LIN {X 0,Y 390.118,Z 257.391,A -85,B 0,C 180,E1 -11800.378,E2 -11800.378} C_VEL
LIN {X 0,Y 390.108,Z 257.393,A -85,B 0,C 180,E1 -11803.544,E2 -11803.544} C_VEL
LIN {X 0,Y 390.089,Z 257.395,A -85,B 0,C 180,E1 -11807.311,E2 -11807.311} C_VEL
LIN {X 0,Y 390.049,Z 257.395,A -85,B 0,C 180,E1 -11811.122,E2 -11811.122} C_VEL
LIN {X 0,Y 390.027,Z 257.402,A -85,B 0,C 180,E1 -11814.484,E2 -11814.484} C_VEL
LIN {X 0,Y 390.06,Z 257.399,A -85,B 0,C 180,E1 -11818.029,E2 -11818.029} C_VEL
LIN {X 0,Y 389.97,Z 257.406,A -85,B 0,C 180,E1 -11820.774,E2 -11820.774} C_VEL
LIN {X 0,Y 389.303,Z 257.492,A -85,B 0,C 180,E1 -11821.636,E2 -11821.636} C_VEL
LIN {X 0,Y 386.453,Z 257.843,A -85,B 0,C 180,E1 -11823.037,E2 -11823.037} C_VEL
LIN {X 0,Y 384.048,Z 258.147,A -85,B 0,C 180,E1 -11824.17,E2 -11824.17} C_VEL
LIN {X 0,Y 383.025,Z 258.271,A -85,B 0,C 180,E1 -11825.046,E2 -11825.046} C_VEL
LIN {X 0,Y 382.946,Z 258.281,A -85,B 0,C 180,E1 -11825.343,E2 -11825.343} C_VEL
LIN {X 0,Y 382.958,Z 258.279,A -85,B 0,C 180,E1 -11828.605,E2 -11828.605} C_VEL
LIN {X 0,Y 382.999,Z 258.276,A -85,B 0,C 180,E1 -11831.344,E2 -11831.344} C_VEL
LIN {X 0,Y 383.025,Z 258.271,A -85,B 0,C 180,E1 -11834.32,E2 -11834.32} C_VEL
LIN {X 0,Y 383.033,Z 258.272,A -85,B 0,C 180,E1 -11837.255,E2 -11837.255} C_VEL
LIN {X 0,Y 382.974,Z 258.276,A -85,B 0,C 180,E1 -11840.42,E2 -11840.42} C_VEL
LIN {X 0,Y 382.987,Z 258.276,A -85,B 0,C 180,E1 -11844.05,E2 -11844.05} C_VEL
LIN {X 0,Y 382.952,Z 258.283,A -85,B 0,C 180,E1 -11847.585,E2 -11847.585} C_VEL
LIN {X 0,Y 382.96,Z 258.278,A -85,B 0,C 180,E1 -11850.306,E2 -11850.306} C_VEL
LIN {X 0,Y 383.052,Z 258.267,A -85,B 0,C 180,E1 -11854.028,E2 -11854.028} C_VEL
LIN {X 0,Y 382.969,Z 258.28,A -85,B 0,C 180,E1 -11857.341,E2 -11857.341} C_VEL
LIN {X 0,Y 383.035,Z 258.274,A -85,B 0,C 180,E1 -11860.723,E2 -11860.723} C_VEL
LIN {X 0,Y 383.059,Z 258.266,A -85,B 0,C 180,E1 -11864.033,E2 -11864.033} C_VEL
LIN {X 0,Y 383.119,Z 258.259,A -85,B 0,C 180,E1 -11867.29,E2 -11867.29} C_VEL
LIN {X 0,Y 383.128,Z 258.263,A -85,B 0,C 180,E1 -11870.504,E2 -11870.504} C_VEL
LIN {X 0,Y 383.248,Z 258.243,A -85,B 0,C 180,E1 -11873.69,E2 -11873.69} C_VEL
LIN {X 0,Y 383.37,Z 258.229,A -85,B 0,C 180,E1 -11877.905,E2 -11877.905} C_VEL
LIN {X 0,Y 383.366,Z 258.233,A -85,B 0,C 180,E1 -11882.107,E2 -11882.107} C_VEL
LIN {X 0,Y 383.229,Z 258.249,A -85,B 0,C 180,E1 -11886.323,E2 -11886.323} C_VEL
LIN {X 0,Y 383.14,Z 258.257,A -85,B 0,C 180,E1 -11889.508,E2 -11889.508} C_VEL
LIN {X 0,Y 383.127,Z 258.26,A -85,B 0,C 180,E1 -11893.541,E2 -11893.541} C_VEL
LIN {X 0,Y 383.056,Z 258.269,A -85,B 0,C 180,E1 -11897.439,E2 -11897.439} C_VEL
LIN {X 0,Y 383.021,Z 258.271,A -85,B 0,C 180,E1 -11900.647,E2 -11900.647} C_VEL
LIN {X 0,Y 383.013,Z 258.276,A -85,B 0,C 180,E1 -11903.814,E2 -11903.814} C_VEL
LIN {X 0,Y 382.976,Z 258.281,A -85,B 0,C 180,E1 -11907.313,E2 -11907.313} C_VEL
LIN {X 0,Y 382.989,Z 258.277,A -85,B 0,C 180,E1 -11910.923,E2 -11910.923} C_VEL
LIN {X 0,Y 383.021,Z 258.276,A -85,B 0,C 180,E1 -11914.673,E2 -11914.673} C_VEL
LIN {X 0,Y 383.005,Z 258.278,A -85,B 0,C 180,E1 -11917.906,E2 -11917.906} C_VEL
LIN {X 0,Y 383.229,Z 259.82,A -85,B 0,C 180,E1 -11919.936,E2 -11919.936} C_VEL
LIN {X 0,Y 383.606,Z 262.486,A -85,B 0,C 180,E1 -11922.877,E2 -11922.877} C_VEL
LIN {X 0,Y 384.023,Z 265.533,A -85,B 0,C 180,E1 -11925.939,E2 -11925.939} C_VEL
LIN {X 0,Y 384.15,Z 268.607,A -85,B 0,C 180,E1 -11928.806,E2 -11928.806} C_VEL
LIN {X 0,Y 383.846,Z 272.282,A -85,B 0,C 180,E1 -11931.94,E2 -11931.94} C_VEL
LIN {X 0,Y 383.375,Z 276.85,A -85,B 0,C 180,E1 -11935.588,E2 -11935.588} C_VEL
LIN {X 0,Y 382.941,Z 281.501,A -85,B 0,C 180,E1 -11939.078,E2 -11939.078} C_VEL
LIN {X 0,Y 382.565,Z 286.485,A -85,B 0,C 180,E1 -11942.661,E2 -11942.661} C_VEL
LIN {X 0,Y 382.195,Z 291.542,A -85,B 0,C 180,E1 -11946.138,E2 -11946.138} C_VEL
LIN {X 0,Y 381.988,Z 297.019,A -85,B 0,C 180,E1 -11949.78,E2 -11949.78} C_VEL
LIN {X 0,Y 381.923,Z 299.239,A -85,B 0,C 180,E1 -11951.102,E2 -11951.102} C_VEL
LIN {X 0,Y 384.001,Z 309.515,A -85,B 0,C 180,E1 -11951.545,E2 -11951.545} C_VEL
LIN {X 0,Y 385.658,Z 318.988,A -85,B 0,C 180,E1 -11952.062,E2 -11952.062} C_VEL
LIN {X 0,Y 387.132,Z 329.109,A -85,B 0,C 180,E1 -11952.736,E2 -11952.736} C_VEL
LIN {X 0,Y 387.167,Z 334.549,A -85,B 0,C 180,E1 -11953.116,E2 -11953.116} C_VEL
LIN {X 0,Y 386.22,Z 345.46,A -85,B 0,C 180,E1 -11954.025,E2 -11954.025} C_VEL
LIN {X 0,Y 385.421,Z 354.407,A -85,B 0,C 180,E1 -11954.94,E2 -11954.94} C_VEL
LIN {X 0,Y 384.666,Z 363.303,A -85,B 0,C 180,E1 -11956.041,E2 -11956.041} C_VEL
LIN {X 0,Y 384.092,Z 370.167,A -85,B 0,C 180,E1 -11957.048,E2 -11957.048} C_VEL
LIN {X 0,Y 383.446,Z 376.37,A -85,B 0,C 180,E1 -11958.101,E2 -11958.101} C_VEL
LIN {X 0,Y 382.875,Z 382.911,A -85,B 0,C 180,E1 -11959.423,E2 -11959.423} C_VEL
LIN {X 0,Y 382.469,Z 387.414,A -85,B 0,C 180,E1 -11960.481,E2 -11960.481} C_VEL
LIN {X 0,Y 382.045,Z 392.908,A -85,B 0,C 180,E1 -11962.07,E2 -11962.07} C_VEL
LIN {X 0,Y 381.783,Z 397.235,A -85,B 0,C 180,E1 -11963.659,E2 -11963.659} C_VEL
LIN {X 0,Y 381.68,Z 399.603,A -85,B 0,C 180,E1 -11964.718,E2 -11964.718} C_VEL
LIN {X 0,Y 381.644,Z 401.403,A -85,B 0,C 180,E1 -11965.776,E2 -11965.776} C_VEL
LIN {X 0,Y 381.564,Z 403.848,A -85,B 0,C 180,E1 -11967.889,E2 -11967.889} C_VEL
LIN {X 0,Y 381.598,Z 404.437,A -85,B 0,C 180,E1 -11968.945,E2 -11968.945} C_VEL
LIN {X 0,Y 381.598,Z 404.437,A -85,B 0,C 180,E1 -11971.055,E2 -11971.055} C_VEL
LIN {X 0,Y 381.564,Z 403.848,A -85,B 0,C 180,E1 -11972.111,E2 -11972.111} C_VEL
LIN {X 0,Y 381.644,Z 401.403,A -85,B 0,C 180,E1 -11974.224,E2 -11974.224} C_VEL
LIN {X 0,Y 381.689,Z 398.553,A -85,B 0,C 180,E1 -11975.768,E2 -11975.768} C_VEL
LIN {X 0,Y 381.947,Z 394.463,A -85,B 0,C 180,E1 -11977.4,E2 -11977.4} C_VEL
LIN {X 0,Y 382.314,Z 389.331,A -85,B 0,C 180,E1 -11978.989,E2 -11978.989} C_VEL
LIN {X 0,Y 382.758,Z 384.067,A -85,B 0,C 180,E1 -11980.313,E2 -11980.313} C_VEL
LIN {X 0,Y 383.294,Z 377.746,A -85,B 0,C 180,E1 -11981.636,E2 -11981.636} C_VEL
LIN {X 0,Y 383.899,Z 371.793,A -85,B 0,C 180,E1 -11982.69,E2 -11982.69} C_VEL
LIN {X 0,Y 384.536,Z 364.863,A -85,B 0,C 180,E1 -11983.744,E2 -11983.744} C_VEL
LIN {X 0,Y 385.231,Z 356.678,A -85,B 0,C 180,E1 -11984.798,E2 -11984.798} C_VEL
LIN {X 0,Y 385.954,Z 348.163,A -85,B 0,C 180,E1 -11985.715,E2 -11985.715} C_VEL
LIN {X 0,Y 386.696,Z 339.445,A -85,B 0,C 180,E1 -11986.497,E2 -11986.497} C_VEL
LIN {X 0,Y 387.344,Z 331.917,A -85,B 0,C 180,E1 -11987.065,E2 -11987.065} C_VEL
LIN {X 0,Y 386.126,Z 321.842,A -85,B 0,C 180,E1 -11987.765,E2 -11987.765} C_VEL
LIN {X 0,Y 384.183,Z 310.483,A -85,B 0,C 180,E1 -11988.408,E2 -11988.408} C_VEL
LIN {X 0,Y 381.981,Z 299.866,A -85,B 0,C 180,E1 -11988.879,E2 -11988.879} C_VEL
LIN {X 0,Y 381.893,Z 299.048,A -85,B 0,C 180,E1 -11988.926,E2 -11988.926} C_VEL
LIN {X 0,Y 382.068,Z 294.919,A -85,B 0,C 180,E1 -11991.585,E2 -11991.585} C_VEL
LIN {X 0,Y 382.33,Z 289.843,A -85,B 0,C 180,E1 -11995.01,E2 -11995.01} C_VEL
LIN {X 0,Y 382.699,Z 284.821,A -85,B 0,C 180,E1 -11998.52,E2 -11998.52} C_VEL
LIN {X 0,Y 382.943,Z 281.501,A -85,B 0,C 180,E1 -12000.921,E2 -12000.921} C_VEL
LIN {X 0,Y 383.405,Z 276.573,A -85,B 0,C 180,E1 -12004.627,E2 -12004.627} C_VEL
LIN {X 0,Y 383.845,Z 272.283,A -85,B 0,C 180,E1 -12008.06,E2 -12008.06} C_VEL
LIN {X 0,Y 384.144,Z 268.607,A -85,B 0,C 180,E1 -12011.194,E2 -12011.194} C_VEL
LIN {X 0,Y 384.185,Z 266.644,A -85,B 0,C 180,E1 -12012.963,E2 -12012.963} C_VEL
LIN {X 0,Y 383.802,Z 263.652,A -85,B 0,C 180,E1 -12015.901,E2 -12015.901} C_VEL
LIN {X 0,Y 383.391,Z 260.995,A -85,B 0,C 180,E1 -12018.726,E2 -12018.726} C_VEL
LIN {X 0,Y 383.005,Z 258.278,A -85,B 0,C 180,E1 -12022.094,E2 -12022.094} C_VEL
LIN {X 0,Y 383.021,Z 258.276,A -85,B 0,C 180,E1 -12025.327,E2 -12025.327} C_VEL
LIN {X 0,Y 382.989,Z 258.277,A -85,B 0,C 180,E1 -12029.077,E2 -12029.077} C_VEL
LIN {X 0,Y 382.976,Z 258.281,A -85,B 0,C 180,E1 -12032.687,E2 -12032.687} C_VEL
LIN {X 0,Y 383.013,Z 258.276,A -85,B 0,C 180,E1 -12036.186,E2 -12036.186} C_VEL
LIN {X 0,Y 383.045,Z 258.268,A -85,B 0,C 180,E1 -12039.593,E2 -12039.593} C_VEL
LIN {X 0,Y 383.072,Z 258.265,A -85,B 0,C 180,E1 -12042.925,E2 -12042.925} C_VEL
LIN {X 0,Y 383.127,Z 258.26,A -85,B 0,C 180,E1 -12046.459,E2 -12046.459} C_VEL
LIN {X 0,Y 383.14,Z 258.257,A -85,B 0,C 180,E1 -12050.492,E2 -12050.492} C_VEL
LIN {X 0,Y 383.229,Z 258.249,A -85,B 0,C 180,E1 -12053.677,E2 -12053.677} C_VEL
LIN {X 0,Y 383.366,Z 258.233,A -85,B 0,C 180,E1 -12057.893,E2 -12057.893} C_VEL
LIN {X 0,Y 383.37,Z 258.229,A -85,B 0,C 180,E1 -12062.095,E2 -12062.095} C_VEL
LIN {X 0,Y 383.228,Z 258.245,A -85,B 0,C 180,E1 -12066.567,E2 -12066.567} C_VEL
LIN {X 0,Y 383.128,Z 258.263,A -85,B 0,C 180,E1 -12069.496,E2 -12069.496} C_VEL
LIN {X 0,Y 383.108,Z 258.264,A -85,B 0,C 180,E1 -12073.529,E2 -12073.529} C_VEL
LIN {X 0,Y 383.073,Z 258.269,A -85,B 0,C 180,E1 -12077.063,E2 -12077.063} C_VEL
LIN {X 0,Y 383.005,Z 258.275,A -85,B 0,C 180,E1 -12080.64,E2 -12080.64} C_VEL
LIN {X 0,Y 382.999,Z 258.274,A -85,B 0,C 180,E1 -12083.801,E2 -12083.801} C_VEL
LIN {X 0,Y 383.051,Z 258.267,A -85,B 0,C 180,E1 -12086.117,E2 -12086.117} C_VEL
LIN {X 0,Y 382.96,Z 258.278,A -85,B 0,C 180,E1 -12089.694,E2 -12089.694} C_VEL
LIN {X 0,Y 382.968,Z 258.278,A -85,B 0,C 180,E1 -12093.395,E2 -12093.395} C_VEL
LIN {X 0,Y 382.994,Z 258.276,A -85,B 0,C 180,E1 -12096.158,E2 -12096.158} C_VEL
LIN {X 0,Y 382.972,Z 258.278,A -85,B 0,C 180,E1 -12099.952,E2 -12099.952} C_VEL
LIN {X 0,Y 383.023,Z 258.273,A -85,B 0,C 180,E1 -12102.783,E2 -12102.783} C_VEL
LIN {X 0,Y 383.027,Z 258.271,A -85,B 0,C 180,E1 -12105.795,E2 -12105.795} C_VEL
LIN {X 0,Y 382.997,Z 258.275,A -85,B 0,C 180,E1 -12108.781,E2 -12108.781} C_VEL
LIN {X 0,Y 382.953,Z 258.285,A -85,B 0,C 180,E1 -12112.091,E2 -12112.091} C_VEL
LIN {X 0,Y 382.966,Z 258.278,A -85,B 0,C 180,E1 -12115.327,E2 -12115.327} C_VEL
LIN {X 0,Y 382.983,Z 258.281,A -85,B 0,C 180,E1 -12117.848,E2 -12117.848} C_VEL
LIN {X 0,Y 383.008,Z 258.277,A -85,B 0,C 180,E1 -12121.717,E2 -12121.717} C_VEL
LIN {X 0,Y 382.997,Z 258.274,A -85,B 0,C 180,E1 -12125.036,E2 -12125.036} C_VEL
LIN {X 0,Y 383.016,Z 258.271,A -85,B 0,C 180,E1 -12128.471,E2 -12128.471} C_VEL
LIN {X 0,Y 383.034,Z 258.274,A -85,B 0,C 180,E1 -12131.825,E2 -12131.825} C_VEL
LIN {X 0,Y 383.055,Z 258.272,A -85,B 0,C 180,E1 -12135.116,E2 -12135.116} C_VEL
LIN {X 0,Y 383.046,Z 258.271,A -85,B 0,C 180,E1 -12138.357,E2 -12138.357} C_VEL
LIN {X 0,Y 383.112,Z 258.465,A -85,B 0,C 180,E1 -12139.597,E2 -12139.597} C_VEL
LIN {X 0,Y 383.808,Z 260.603,A -85,B 0,C 180,E1 -12139.949,E2 -12139.949} C_VEL
LIN {X 0,Y 385.342,Z 262.607,A -85,B 0,C 180,E1 -12140.685,E2 -12140.685} C_VEL
LIN {X 0,Y 387.431,Z 263.893,A -85,B 0,C 180,E1 -12141.656,E2 -12141.656} C_VEL
LIN {X 0,Y 388.82,Z 264.575,A -85,B 0,C 180,E1 -12142.393,E2 -12142.393} C_VEL
LIN {X 0,Y 389.855,Z 266.733,A -85,B 0,C 180,E1 -12143.075,E2 -12143.075} C_VEL
LIN {X 0,Y 391.629,Z 268.873,A -85,B 0,C 180,E1 -12144.336,E2 -12144.336} C_VEL
LIN {X 0,Y 393.42,Z 270.078,A -85,B 0,C 180,E1 -12145.902,E2 -12145.902} C_VEL
LIN {X 0,Y 394.315,Z 270.312,A -85,B 0,C 180,E1 -12146.935,E2 -12146.935} C_VEL
LIN {X 0,Y 395.344,Z 270.546,A -85,B 0,C 180,E1 -12148.981,E2 -12148.981} C_VEL
LIN {X 0,Y 395.505,Z 270.523,A -85,B 0,C 180,E1 -12150,E2 -12150} C_VEL
LIN {X 0,Y 394.942,Z 270.448,A -85,B 0,C 180,E1 -12152.04,E2 -12152.04} C_VEL
LIN {X 0,Y 394.144,Z 270.274,A -85,B 0,C 180,E1 -12153.268,E2 -12153.268} C_VEL
LIN {X 0,Y 392.863,Z 269.796,A -85,B 0,C 180,E1 -12154.617,E2 -12154.617} C_VEL
LIN {X 0,Y 390.976,Z 268.254,A -85,B 0,C 180,E1 -12156.127,E2 -12156.127} C_VEL
LIN {X 0,Y 389.275,Z 265.68,A -85,B 0,C 180,E1 -12157.318,E2 -12157.318} C_VEL
LIN {X 0,Y 388.598,Z 264.268,A -85,B 0,C 180,E1 -12157.735,E2 -12157.735} C_VEL
LIN {X 0,Y 386.111,Z 263.182,A -85,B 0,C 180,E1 -12158.966,E2 -12158.966} C_VEL
LIN {X 0,Y 384.201,Z 261.281,A -85,B 0,C 180,E1 -12159.861,E2 -12159.861} C_VEL
LIN {X 0,Y 383.227,Z 259.103,A -85,B 0,C 180,E1 -12160.333,E2 -12160.333} C_VEL
LIN {X 0,Y 383.073,Z 258.269,A -85,B 0,C 180,E1 -12160.438,E2 -12160.438} C_VEL
LIN {X 0,Y 383.066,Z 258.269,A -85,B 0,C 180,E1 -12163.798,E2 -12163.798} C_VEL
LIN {X 0,Y 383.036,Z 258.273,A -85,B 0,C 180,E1 -12167.458,E2 -12167.458} C_VEL
LIN {X 0,Y 383.005,Z 258.276,A -85,B 0,C 180,E1 -12170.664,E2 -12170.664} C_VEL
LIN {X 0,Y 382.99,Z 258.276,A -85,B 0,C 180,E1 -12173.81,E2 -12173.81} C_VEL
LIN {X 0,Y 383,Z 258.273,A -85,B 0,C 180,E1 -12177.306,E2 -12177.306} C_VEL
LIN {X 0,Y 382.941,Z 258.281,A -85,B 0,C 180,E1 -12180.922,E2 -12180.922} C_VEL
LIN {X 0,Y 382.965,Z 258.28,A -85,B 0,C 180,E1 -12184.344,E2 -12184.344} C_VEL
LIN {X 0,Y 382.946,Z 258.281,A -85,B 0,C 180,E1 -12185.343,E2 -12185.343} C_VEL
LIN {X 0,Y 382.302,Z 258.367,A -85,B 0,C 180,E1 -12186.221,E2 -12186.221} C_VEL
LIN {X 0,Y 379.489,Z 258.724,A -85,B 0,C 180,E1 -12187.65,E2 -12187.65} C_VEL
LIN {X 0,Y 377.089,Z 259.023,A -85,B 0,C 180,E1 -12188.804,E2 -12188.804} C_VEL
LIN {X 0,Y 376.043,Z 259.147,A -85,B 0,C 180,E1 -12189.697,E2 -12189.697} C_VEL
LIN {X 0,Y 375.949,Z 259.156,A -85,B 0,C 180,E1 -12189.999,E2 -12189.999} C_VEL
LIN {X 0,Y 375.956,Z 259.157,A -85,B 0,C 180,E1 -12193.761,E2 -12193.761} C_VEL
LIN {X 0,Y 375.955,Z 259.151,A -85,B 0,C 180,E1 -12196.806,E2 -12196.806} C_VEL
LIN {X 0,Y 375.951,Z 259.153,A -85,B 0,C 180,E1 -12200.035,E2 -12200.035} C_VEL
LIN {X 0,Y 375.926,Z 259.16,A -85,B 0,C 180,E1 -12203.502,E2 -12203.502} C_VEL
LIN {X 0,Y 375.924,Z 259.156,A -85,B 0,C 180,E1 -12205.895,E2 -12205.895} C_VEL
LIN {X 0,Y 375.932,Z 259.156,A -85,B 0,C 180,E1 -12209.694,E2 -12209.694} C_VEL
LIN {X 0,Y 375.991,Z 259.15,A -85,B 0,C 180,E1 -12213.354,E2 -12213.354} C_VEL
LIN {X 0,Y 375.957,Z 259.156,A -85,B 0,C 180,E1 -12216.894,E2 -12216.894} C_VEL
LIN {X 0,Y 375.973,Z 259.15,A -85,B 0,C 180,E1 -12220.346,E2 -12220.346} C_VEL
LIN {X 0,Y 376.004,Z 259.145,A -85,B 0,C 180,E1 -12223.725,E2 -12223.725} C_VEL
LIN {X 0,Y 376.086,Z 259.137,A -85,B 0,C 180,E1 -12227.049,E2 -12227.049} C_VEL
LIN {X 0,Y 376.098,Z 259.137,A -85,B 0,C 180,E1 -12230.325,E2 -12230.325} C_VEL
LIN {X 0,Y 376.207,Z 259.12,A -85,B 0,C 180,E1 -12233.571,E2 -12233.571} C_VEL
LIN {X 0,Y 376.335,Z 259.105,A -85,B 0,C 180,E1 -12237.866,E2 -12237.866} C_VEL
LIN {X 0,Y 376.331,Z 259.109,A -85,B 0,C 180,E1 -12242.147,E2 -12242.147} C_VEL
LIN {X 0,Y 376.189,Z 259.125,A -85,B 0,C 180,E1 -12246.442,E2 -12246.442} C_VEL
LIN {X 0,Y 376.111,Z 259.134,A -85,B 0,C 180,E1 -12249.687,E2 -12249.687} C_VEL
LIN {X 0,Y 376.092,Z 259.138,A -85,B 0,C 180,E1 -12253.663,E2 -12253.663} C_VEL
LIN {X 0,Y 376.01,Z 259.148,A -85,B 0,C 180,E1 -12257.594,E2 -12257.594} C_VEL
LIN {X 0,Y 375.984,Z 259.147,A -85,B 0,C 180,E1 -12260.837,E2 -12260.837} C_VEL
LIN {X 0,Y 375.941,Z 259.153,A -85,B 0,C 180,E1 -12264.29,E2 -12264.29} C_VEL
LIN {X 0,Y 375.918,Z 259.156,A -85,B 0,C 180,E1 -12266.665,E2 -12266.665} C_VEL
LIN {X 0,Y 375.921,Z 259.158,A -85,B 0,C 180,E1 -12269.088,E2 -12269.088} C_VEL
LIN {X 0,Y 375.964,Z 259.154,A -85,B 0,C 180,E1 -12271.566,E2 -12271.566} C_VEL
LIN {X 0,Y 375.959,Z 259.156,A -85,B 0,C 180,E1 -12275.42,E2 -12275.42} C_VEL
LIN {X 0,Y 375.993,Z 259.438,A -85,B 0,C 180,E1 -12278.09,E2 -12278.09} C_VEL
LIN {X 0,Y 376.435,Z 262.515,A -85,B 0,C 180,E1 -12281.688,E2 -12281.688} C_VEL
LIN {X 0,Y 376.894,Z 265.773,A -85,B 0,C 180,E1 -12285.126,E2 -12285.126} C_VEL
LIN {X 0,Y 377.133,Z 268.951,A -85,B 0,C 180,E1 -12288.2,E2 -12288.2} C_VEL
LIN {X 0,Y 376.877,Z 272.763,A -85,B 0,C 180,E1 -12291.562,E2 -12291.562} C_VEL
LIN {X 0,Y 376.351,Z 277.292,A -85,B 0,C 180,E1 -12295.257,E2 -12295.257} C_VEL
LIN {X 0,Y 375.939,Z 281.396,A -85,B 0,C 180,E1 -12298.437,E2 -12298.437} C_VEL
LIN {X 0,Y 375.617,Z 285.627,A -85,B 0,C 180,E1 -12301.576,E2 -12301.576} C_VEL
LIN {X 0,Y 375.317,Z 289.711,A -85,B 0,C 180,E1 -12304.489,E2 -12304.489} C_VEL
LIN {X 0,Y 374.996,Z 294.771,A -85,B 0,C 180,E1 -12307.987,E2 -12307.987} C_VEL
LIN {X 0,Y 374.848,Z 298.856,A -85,B 0,C 180,E1 -12310.723,E2 -12310.723} C_VEL
LIN {X 0,Y 377.05,Z 309.739,A -85,B 0,C 180,E1 -12311.21,E2 -12311.21} C_VEL
LIN {X 0,Y 378.634,Z 318.769,A -85,B 0,C 180,E1 -12311.718,E2 -12311.718} C_VEL
LIN {X 0,Y 379.938,Z 327.831,A -85,B 0,C 180,E1 -12312.326,E2 -12312.326} C_VEL
LIN {X 0,Y 380.449,Z 333.165,A -85,B 0,C 180,E1 -12312.717,E2 -12312.717} C_VEL
LIN {X 0,Y 379.383,Z 345.248,A -85,B 0,C 180,E1 -12313.729,E2 -12313.729} C_VEL
LIN {X 0,Y 378.529,Z 354.195,A -85,B 0,C 180,E1 -12314.659,E2 -12314.659} C_VEL
LIN {X 0,Y 377.887,Z 361.899,A -85,B 0,C 180,E1 -12315.615,E2 -12315.615} C_VEL
LIN {X 0,Y 377.16,Z 369.955,A -85,B 0,C 180,E1 -12316.805,E2 -12316.805} C_VEL
LIN {X 0,Y 376.482,Z 376.158,A -85,B 0,C 180,E1 -12317.877,E2 -12317.877} C_VEL
LIN {X 0,Y 375.842,Z 382.698,A -85,B 0,C 180,E1 -12319.223,E2 -12319.223} C_VEL
LIN {X 0,Y 375.455,Z 387.202,A -85,B 0,C 180,E1 -12320.301,E2 -12320.301} C_VEL
LIN {X 0,Y 374.976,Z 392.696,A -85,B 0,C 180,E1 -12321.919,E2 -12321.919} C_VEL
LIN {X 0,Y 374.7,Z 397.023,A -85,B 0,C 180,E1 -12323.538,E2 -12323.538} C_VEL
LIN {X 0,Y 374.588,Z 399.391,A -85,B 0,C 180,E1 -12324.617,E2 -12324.617} C_VEL
LIN {X 0,Y 374.571,Z 401.192,A -85,B 0,C 180,E1 -12325.696,E2 -12325.696} C_VEL
LIN {X 0,Y 374.463,Z 403.636,A -85,B 0,C 180,E1 -12327.849,E2 -12327.849} C_VEL
LIN {X 0,Y 374.499,Z 404.226,A -85,B 0,C 180,E1 -12328.925,E2 -12328.925} C_VEL
LIN {X 0,Y 374.499,Z 404.226,A -85,B 0,C 180,E1 -12331.075,E2 -12331.075} C_VEL
LIN {X 0,Y 374.463,Z 403.636,A -85,B 0,C 180,E1 -12332.151,E2 -12332.151} C_VEL
LIN {X 0,Y 374.571,Z 401.192,A -85,B 0,C 180,E1 -12334.304,E2 -12334.304} C_VEL
LIN {X 0,Y 374.588,Z 399.391,A -85,B 0,C 180,E1 -12335.383,E2 -12335.383} C_VEL
LIN {X 0,Y 374.784,Z 395.782,A -85,B 0,C 180,E1 -12337.001,E2 -12337.001} C_VEL
LIN {X 0,Y 375.113,Z 391.035,A -85,B 0,C 180,E1 -12338.62,E2 -12338.62} C_VEL
LIN {X 0,Y 375.629,Z 385.01,A -85,B 0,C 180,E1 -12340.238,E2 -12340.238} C_VEL
LIN {X 0,Y 376.189,Z 378.91,A -85,B 0,C 180,E1 -12341.585,E2 -12341.585} C_VEL
LIN {X 0,Y 376.798,Z 373.209,A -85,B 0,C 180,E1 -12342.659,E2 -12342.659} C_VEL
LIN {X 0,Y 377.599,Z 364.65,A -85,B 0,C 180,E1 -12344.002,E2 -12344.002} C_VEL
LIN {X 0,Y 378.319,Z 356.465,A -85,B 0,C 180,E1 -12345.074,E2 -12345.074} C_VEL
LIN {X 0,Y 379.121,Z 347.952,A -85,B 0,C 180,E1 -12346.006,E2 -12346.006} C_VEL
LIN {X 0,Y 379.875,Z 339.233,A -85,B 0,C 180,E1 -12346.802,E2 -12346.802} C_VEL
LIN {X 0,Y 380.438,Z 331.844,A -85,B 0,C 180,E1 -12347.375,E2 -12347.375} C_VEL
LIN {X 0,Y 378.944,Z 320.564,A -85,B 0,C 180,E1 -12348.17,E2 -12348.17} C_VEL
LIN {X 0,Y 377.148,Z 310.281,A -85,B 0,C 180,E1 -12348.763,E2 -12348.763} C_VEL
LIN {X 0,Y 374.932,Z 299.685,A -85,B 0,C 180,E1 -12349.246,E2 -12349.246} C_VEL
LIN {X 0,Y 374.855,Z 298.829,A -85,B 0,C 180,E1 -12349.295,E2 -12349.295} C_VEL
LIN {X 0,Y 375.109,Z 292.812,A -85,B 0,C 180,E1 -12353.349,E2 -12353.349} C_VEL
LIN {X 0,Y 375.402,Z 288.027,A -85,B 0,C 180,E1 -12356.699,E2 -12356.699} C_VEL
LIN {X 0,Y 375.836,Z 283.042,A -85,B 0,C 180,E1 -12360.323,E2 -12360.323} C_VEL
LIN {X 0,Y 376.255,Z 278.125,A -85,B 0,C 180,E1 -12364.08,E2 -12364.08} C_VEL
LIN {X 0,Y 376.624,Z 274.901,A -85,B 0,C 180,E1 -12366.664,E2 -12366.664} C_VEL
LIN {X 0,Y 376.967,Z 271.718,A -85,B 0,C 180,E1 -12369.336,E2 -12369.336} C_VEL
LIN {X 0,Y 377.153,Z 268.57,A -85,B 0,C 180,E1 -12372.131,E2 -12372.131} C_VEL
LIN {X 0,Y 376.914,Z 265.734,A -85,B 0,C 180,E1 -12374.877,E2 -12374.877} C_VEL
LIN {X 0,Y 376.433,Z 262.513,A -85,B 0,C 180,E1 -12378.313,E2 -12378.313} C_VEL
LIN {X 0,Y 375.993,Z 259.442,A -85,B 0,C 180,E1 -12381.91,E2 -12381.91} C_VEL
LIN {X 0,Y 375.959,Z 259.155,A -85,B 0,C 180,E1 -12384.58,E2 -12384.58} C_VEL
LIN {X 0,Y 375.964,Z 259.154,A -85,B 0,C 180,E1 -12388.434,E2 -12388.434} C_VEL
LIN {X 0,Y 375.925,Z 259.157,A -85,B 0,C 180,E1 -12392.13,E2 -12392.13} C_VEL
LIN {X 0,Y 375.943,Z 259.158,A -85,B 0,C 180,E1 -12394.529,E2 -12394.529} C_VEL
LIN {X 0,Y 375.976,Z 259.15,A -85,B 0,C 180,E1 -12396.882,E2 -12396.882} C_VEL
LIN {X 0,Y 375.978,Z 259.154,A -85,B 0,C 180,E1 -12400.333,E2 -12400.333} C_VEL
LIN {X 0,Y 375.977,Z 259.15,A -85,B 0,C 180,E1 -12403.711,E2 -12403.711} C_VEL
LIN {X 0,Y 376.104,Z 259.132,A -85,B 0,C 180,E1 -12407.036,E2 -12407.036} C_VEL
LIN {X 0,Y 376.111,Z 259.134,A -85,B 0,C 180,E1 -12410.313,E2 -12410.313} C_VEL
LIN {X 0,Y 376.189,Z 259.125,A -85,B 0,C 180,E1 -12413.558,E2 -12413.558} C_VEL
LIN {X 0,Y 376.331,Z 259.109,A -85,B 0,C 180,E1 -12417.853,E2 -12417.853} C_VEL
LIN {X 0,Y 376.335,Z 259.105,A -85,B 0,C 180,E1 -12422.134,E2 -12422.134} C_VEL
LIN {X 0,Y 376.195,Z 259.121,A -85,B 0,C 180,E1 -12426.554,E2 -12426.554} C_VEL
LIN {X 0,Y 376.098,Z 259.137,A -85,B 0,C 180,E1 -12429.675,E2 -12429.675} C_VEL
LIN {X 0,Y 376.072,Z 259.139,A -85,B 0,C 180,E1 -12433.651,E2 -12433.651} C_VEL
LIN {X 0,Y 376.011,Z 259.148,A -85,B 0,C 180,E1 -12437.393,E2 -12437.393} C_VEL
LIN {X 0,Y 375.955,Z 259.155,A -85,B 0,C 180,E1 -12440.825,E2 -12440.825} C_VEL
LIN {X 0,Y 375.963,Z 259.151,A -85,B 0,C 180,E1 -12444.275,E2 -12444.275} C_VEL
LIN {X 0,Y 375.991,Z 259.15,A -85,B 0,C 180,E1 -12446.646,E2 -12446.646} C_VEL
LIN {X 0,Y 375.932,Z 259.156,A -85,B 0,C 180,E1 -12450.306,E2 -12450.306} C_VEL
LIN {X 0,Y 375.924,Z 259.156,A -85,B 0,C 180,E1 -12454.105,E2 -12454.105} C_VEL
LIN {X 0,Y 375.915,Z 259.161,A -85,B 0,C 180,E1 -12456.735,E2 -12456.735} C_VEL
LIN {X 0,Y 375.951,Z 259.153,A -85,B 0,C 180,E1 -12459.965,E2 -12459.965} C_VEL
LIN {X 0,Y 375.955,Z 259.152,A -85,B 0,C 180,E1 -12463.75,E2 -12463.75} C_VEL
LIN {X 0,Y 375.954,Z 259.153,A -85,B 0,C 180,E1 -12466.795,E2 -12466.795} C_VEL
LIN {X 0,Y 375.95,Z 259.156,A -85,B 0,C 180,E1 -12470.022,E2 -12470.022} C_VEL
LIN {X 0,Y 375.914,Z 259.157,A -85,B 0,C 180,E1 -12473.491,E2 -12473.491} C_VEL
LIN {X 0,Y 375.909,Z 259.162,A -85,B 0,C 180,E1 -12475.884,E2 -12475.884} C_VEL
LIN {X 0,Y 375.914,Z 259.16,A -85,B 0,C 180,E1 -12479.684,E2 -12479.684} C_VEL
LIN {X 0,Y 375.946,Z 259.155,A -85,B 0,C 180,E1 -12482.138,E2 -12482.138} C_VEL
LIN {X 0,Y 375.95,Z 259.152,A -85,B 0,C 180,E1 -12484.535,E2 -12484.535} C_VEL
LIN {X 0,Y 375.966,Z 259.152,A -85,B 0,C 180,E1 -12488.046,E2 -12488.046} C_VEL
LIN {X 0,Y 375.972,Z 259.154,A -85,B 0,C 180,E1 -12491.472,E2 -12491.472} C_VEL
LIN {X 0,Y 376.003,Z 259.15,A -85,B 0,C 180,E1 -12494.831,E2 -12494.831} C_VEL
LIN {X 0,Y 376.055,Z 259.145,A -85,B 0,C 180,E1 -12497.281,E2 -12497.281} C_VEL
LIN {X 0,Y 376.671,Z 261.359,A -85,B 0,C 180,E1 -12497.576,E2 -12497.576} C_VEL
LIN {X 0,Y 378.386,Z 263.615,A -85,B 0,C 180,E1 -12498.211,E2 -12498.211} C_VEL
LIN {X 0,Y 380.852,Z 265.017,A -85,B 0,C 180,E1 -12499.097,E2 -12499.097} C_VEL
LIN {X 0,Y 381.337,Z 265.87,A -85,B 0,C 180,E1 -12499.313,E2 -12499.313} C_VEL
LIN {X 0,Y 382.811,Z 268.253,A -85,B 0,C 180,E1 -12499.956,E2 -12499.956} C_VEL
LIN {X 0,Y 385.297,Z 270.371,A -85,B 0,C 180,E1 -12501.081,E2 -12501.081} C_VEL
LIN {X 0,Y 387.386,Z 271.48,A -85,B 0,C 180,E1 -12502.118,E2 -12502.118} C_VEL
LIN {X 0,Y 389.029,Z 274.176,A -85,B 0,C 180,E1 -12503.143,E2 -12503.143} C_VEL
LIN {X 0,Y 390.886,Z 276.096,A -85,B 0,C 180,E1 -12504.454,E2 -12504.454} C_VEL
LIN {X 0,Y 392.53,Z 277.121,A -85,B 0,C 180,E1 -12505.893,E2 -12505.893} C_VEL
LIN {X 0,Y 394.08,Z 277.498,A -85,B 0,C 180,E1 -12507.956,E2 -12507.956} C_VEL
LIN {X 0,Y 394.642,Z 277.554,A -85,B 0,C 180,E1 -12510,E2 -12510} C_VEL
LIN {X 0,Y 394.08,Z 277.495,A -85,B 0,C 180,E1 -12512.044,E2 -12512.044} C_VEL
LIN {X 0,Y 392.53,Z 277.122,A -85,B 0,C 180,E1 -12514.107,E2 -12514.107} C_VEL
LIN {X 0,Y 390.526,Z 275.818,A -85,B 0,C 180,E1 -12515.81,E2 -12515.81} C_VEL
LIN {X 0,Y 388.468,Z 273.378,A -85,B 0,C 180,E1 -12517.227,E2 -12517.227} C_VEL
LIN {X 0,Y 387.164,Z 271.164,A -85,B 0,C 180,E1 -12518.013,E2 -12518.013} C_VEL
LIN {X 0,Y 384.483,Z 269.856,A -85,B 0,C 180,E1 -12519.283,E2 -12519.283} C_VEL
LIN {X 0,Y 382.311,Z 267.587,A -85,B 0,C 180,E1 -12520.258,E2 -12520.258} C_VEL
LIN {X 0,Y 380.988,Z 265.059,A -85,B 0,C 180,E1 -12520.852,E2 -12520.852} C_VEL
LIN {X 0,Y 378.578,Z 263.789,A -85,B 0,C 180,E1 -12521.722,E2 -12521.722} C_VEL
LIN {X 0,Y 376.761,Z 261.555,A -85,B 0,C 180,E1 -12522.387,E2 -12522.387} C_VEL
LIN {X 0,Y 376.086,Z 259.512,A -85,B 0,C 180,E1 -12522.684,E2 -12522.684} C_VEL
LIN {X 0,Y 376.031,Z 259.147,A -85,B 0,C 180,E1 -12522.754,E2 -12522.754} C_VEL
LIN {X 0,Y 375.972,Z 259.154,A -85,B 0,C 180,E1 -12526.283,E2 -12526.283} C_VEL
LIN {X 0,Y 375.958,Z 259.153,A -85,B 0,C 180,E1 -12529.662,E2 -12529.662} C_VEL
LIN {X 0,Y 375.972,Z 259.149,A -85,B 0,C 180,E1 -12533.113,E2 -12533.113} C_VEL
LIN {X 0,Y 375.963,Z 259.152,A -85,B 0,C 180,E1 -12536.656,E2 -12536.656} C_VEL
LIN {X 0,Y 375.921,Z 259.155,A -85,B 0,C 180,E1 -12539.083,E2 -12539.083} C_VEL
LIN {X 0,Y 375.903,Z 259.158,A -85,B 0,C 180,E1 -12542.832,E2 -12542.832} C_VEL
LIN {X 0,Y 375.906,Z 259.158,A -85,B 0,C 180,E1 -12545.42,E2 -12545.42} C_VEL
LIN {X 0,Y 375.928,Z 259.157,A -85,B 0,C 180,E1 -12548.276,E2 -12548.276} C_VEL
LIN {X 0,Y 375.949,Z 259.156,A -85,B 0,C 180,E1 -12549.999,E2 -12549.999} C_VEL
LIN {X 0,Y 375.255,Z 259.239,A -85,B 0,C 180,E1 -12550.893,E2 -12550.893} C_VEL
LIN {X 0,Y 372.382,Z 259.597,A -85,B 0,C 180,E1 -12552.346,E2 -12552.346} C_VEL
LIN {X 0,Y 369.99,Z 259.898,A -85,B 0,C 180,E1 -12553.521,E2 -12553.521} C_VEL
LIN {X 0,Y 369.001,Z 260.018,A -85,B 0,C 180,E1 -12554.43,E2 -12554.43} C_VEL
LIN {X 0,Y 368.94,Z 260.025,A -85,B 0,C 180,E1 -12554.737,E2 -12554.737} C_VEL
LIN {X 0,Y 368.898,Z 260.031,A -85,B 0,C 180,E1 -12558.191,E2 -12558.191} C_VEL
LIN {X 0,Y 368.867,Z 260.039,A -85,B 0,C 180,E1 -12561.366,E2 -12561.366} C_VEL
LIN {X 0,Y 368.9,Z 260.034,A -85,B 0,C 180,E1 -12565.153,E2 -12565.153} C_VEL
LIN {X 0,Y 368.897,Z 260.034,A -85,B 0,C 180,E1 -12569.053,E2 -12569.053} C_VEL
LIN {X 0,Y 368.934,Z 260.029,A -85,B 0,C 180,E1 -12572.803,E2 -12572.803} C_VEL
LIN {X 0,Y 368.91,Z 260.029,A -85,B 0,C 180,E1 -12576.123,E2 -12576.123} C_VEL
LIN {X 0,Y 368.906,Z 260.029,A -85,B 0,C 180,E1 -12579.953,E2 -12579.953} C_VEL
LIN {X 0,Y 368.947,Z 260.025,A -85,B 0,C 180,E1 -12583.405,E2 -12583.405} C_VEL
LIN {X 0,Y 369.041,Z 260.018,A -85,B 0,C 180,E1 -12586.797,E2 -12586.797} C_VEL
LIN {X 0,Y 369.048,Z 260.013,A -85,B 0,C 180,E1 -12590.138,E2 -12590.138} C_VEL
LIN {X 0,Y 369.167,Z 259.996,A -85,B 0,C 180,E1 -12593.448,E2 -12593.448} C_VEL
LIN {X 0,Y 369.299,Z 259.981,A -85,B 0,C 180,E1 -12597.825,E2 -12597.825} C_VEL
LIN {X 0,Y 369.295,Z 259.986,A -85,B 0,C 180,E1 -12602.188,E2 -12602.188} C_VEL
LIN {X 0,Y 369.151,Z 260,A -85,B 0,C 180,E1 -12606.565,E2 -12606.565} C_VEL
LIN {X 0,Y 369.061,Z 260.014,A -85,B 0,C 180,E1 -12609.874,E2 -12609.874} C_VEL
LIN {X 0,Y 369.039,Z 260.017,A -85,B 0,C 180,E1 -12613.778,E2 -12613.778} C_VEL
LIN {X 0,Y 368.957,Z 260.029,A -85,B 0,C 180,E1 -12617.75,E2 -12617.75} C_VEL
LIN {X 0,Y 368.914,Z 260.03,A -85,B 0,C 180,E1 -12621.226,E2 -12621.226} C_VEL
LIN {X 0,Y 368.914,Z 260.031,A -85,B 0,C 180,E1 -12623.878,E2 -12623.878} C_VEL
LIN {X 0,Y 368.865,Z 260.038,A -85,B 0,C 180,E1 -12627.217,E2 -12627.217} C_VEL
LIN {X 0,Y 368.901,Z 260.033,A -85,B 0,C 180,E1 -12629.697,E2 -12629.697} C_VEL
LIN {X 0,Y 368.906,Z 260.032,A -85,B 0,C 180,E1 -12633.047,E2 -12633.047} C_VEL
LIN {X 0,Y 368.921,Z 260.031,A -85,B 0,C 180,E1 -12636.202,E2 -12636.202} C_VEL
LIN {X 0,Y 368.923,Z 260.206,A -85,B 0,C 180,E1 -12637.566,E2 -12637.566} C_VEL
LIN {X 0,Y 369.251,Z 262.54,A -85,B 0,C 180,E1 -12640.42,E2 -12640.42} C_VEL
LIN {X 0,Y 369.704,Z 265.523,A -85,B 0,C 180,E1 -12643.75,E2 -12643.75} C_VEL
LIN {X 0,Y 370.041,Z 268.578,A -85,B 0,C 180,E1 -12646.865,E2 -12646.865} C_VEL
LIN {X 0,Y 370.001,Z 271.691,A -85,B 0,C 180,E1 -12649.774,E2 -12649.774} C_VEL
LIN {X 0,Y 369.604,Z 275.406,A -85,B 0,C 180,E1 -12653.005,E2 -12653.005} C_VEL
LIN {X 0,Y 369.111,Z 279.672,A -85,B 0,C 180,E1 -12656.485,E2 -12656.485} C_VEL
LIN {X 0,Y 368.836,Z 282.932,A -85,B 0,C 180,E1 -12659.038,E2 -12659.038} C_VEL
LIN {X 0,Y 368.396,Z 287.893,A -85,B 0,C 180,E1 -12662.752,E2 -12662.752} C_VEL
LIN {X 0,Y 368.031,Z 293.03,A -85,B 0,C 180,E1 -12666.444,E2 -12666.444} C_VEL
LIN {X 0,Y 367.773,Z 298.609,A -85,B 0,C 180,E1 -12670.318,E2 -12670.318} C_VEL
LIN {X 0,Y 370.854,Z 313.837,A -85,B 0,C 180,E1 -12671.063,E2 -12671.063} C_VEL
LIN {X 0,Y 372.829,Z 326.677,A -85,B 0,C 180,E1 -12671.912,E2 -12671.912} C_VEL
LIN {X 0,Y 373.571,Z 334.125,A -85,B 0,C 180,E1 -12672.482,E2 -12672.482} C_VEL
LIN {X 0,Y 372.565,Z 345.036,A -85,B 0,C 180,E1 -12673.423,E2 -12673.423} C_VEL
LIN {X 0,Y 371.675,Z 353.983,A -85,B 0,C 180,E1 -12674.369,E2 -12674.369} C_VEL
LIN {X 0,Y 370.948,Z 362.056,A -85,B 0,C 180,E1 -12675.394,E2 -12675.394} C_VEL
LIN {X 0,Y 370.231,Z 369.743,A -85,B 0,C 180,E1 -12676.554,E2 -12676.554} C_VEL
LIN {X 0,Y 369.53,Z 375.946,A -85,B 0,C 180,E1 -12677.646,E2 -12677.646} C_VEL
LIN {X 0,Y 368.82,Z 382.485,A -85,B 0,C 180,E1 -12679.015,E2 -12679.015} C_VEL
LIN {X 0,Y 368.417,Z 386.99,A -85,B 0,C 180,E1 -12680.114,E2 -12680.114} C_VEL
LIN {X 0,Y 367.923,Z 392.484,A -85,B 0,C 180,E1 -12681.763,E2 -12681.763} C_VEL
LIN {X 0,Y 367.616,Z 396.811,A -85,B 0,C 180,E1 -12683.413,E2 -12683.413} C_VEL
LIN {X 0,Y 367.503,Z 399.179,A -85,B 0,C 180,E1 -12684.513,E2 -12684.513} C_VEL
LIN {X 0,Y 367.478,Z 400.98,A -85,B 0,C 180,E1 -12685.613,E2 -12685.613} C_VEL
LIN {X 0,Y 367.365,Z 403.425,A -85,B 0,C 180,E1 -12687.807,E2 -12687.807} C_VEL
LIN {X 0,Y 367.4,Z 404.015,A -85,B 0,C 180,E1 -12688.904,E2 -12688.904} C_VEL
LIN {X 0,Y 367.4,Z 404.015,A -85,B 0,C 180,E1 -12691.096,E2 -12691.096} C_VEL
LIN {X 0,Y 367.365,Z 403.425,A -85,B 0,C 180,E1 -12692.193,E2 -12692.193} C_VEL
LIN {X 0,Y 367.478,Z 400.98,A -85,B 0,C 180,E1 -12694.387,E2 -12694.387} C_VEL
LIN {X 0,Y 367.545,Z 397.923,A -85,B 0,C 180,E1 -12696.084,E2 -12696.084} C_VEL
LIN {X 0,Y 367.806,Z 394.038,A -85,B 0,C 180,E1 -12697.686,E2 -12697.686} C_VEL
LIN {X 0,Y 368.239,Z 388.907,A -85,B 0,C 180,E1 -12699.336,E2 -12699.336} C_VEL
LIN {X 0,Y 368.742,Z 383.642,A -85,B 0,C 180,E1 -12700.709,E2 -12700.709} C_VEL
LIN {X 0,Y 369.352,Z 377.322,A -85,B 0,C 180,E1 -12702.082,E2 -12702.082} C_VEL
LIN {X 0,Y 370.014,Z 371.369,A -85,B 0,C 180,E1 -12703.175,E2 -12703.175} C_VEL
LIN {X 0,Y 370.809,Z 363.251,A -85,B 0,C 180,E1 -12704.437,E2 -12704.437} C_VEL
LIN {X 0,Y 371.525,Z 355.117,A -85,B 0,C 180,E1 -12705.497,E2 -12705.497} C_VEL
LIN {X 0,Y 372.422,Z 346.388,A -85,B 0,C 180,E1 -12706.443,E2 -12706.443} C_VEL
LIN {X 0,Y 373.238,Z 337.39,A -85,B 0,C 180,E1 -12707.251,E2 -12707.251} C_VEL
LIN {X 0,Y 373.452,Z 331.756,A -85,B 0,C 180,E1 -12707.701,E2 -12707.701} C_VEL
LIN {X 0,Y 371.994,Z 320.816,A -85,B 0,C 180,E1 -12708.496,E2 -12708.496} C_VEL
LIN {X 0,Y 370.109,Z 309.943,A -85,B 0,C 180,E1 -12709.138,E2 -12709.138} C_VEL
LIN {X 0,Y 367.837,Z 299.377,A -85,B 0,C 180,E1 -12709.635,E2 -12709.635} C_VEL
LIN {X 0,Y 367.776,Z 298.614,A -85,B 0,C 180,E1 -12709.678,E2 -12709.678} C_VEL
LIN {X 0,Y 368.036,Z 292.909,A -85,B 0,C 180,E1 -12713.641,E2 -12713.641} C_VEL
LIN {X 0,Y 368.396,Z 287.893,A -85,B 0,C 180,E1 -12717.248,E2 -12717.248} C_VEL
LIN {X 0,Y 368.836,Z 282.932,A -85,B 0,C 180,E1 -12720.962,E2 -12720.962} C_VEL
LIN {X 0,Y 369.341,Z 278.05,A -85,B 0,C 180,E1 -12724.809,E2 -12724.809} C_VEL
LIN {X 0,Y 369.664,Z 274.838,A -85,B 0,C 180,E1 -12727.472,E2 -12727.472} C_VEL
LIN {X 0,Y 370.025,Z 271.305,A -85,B 0,C 180,E1 -12730.554,E2 -12730.554} C_VEL
LIN {X 0,Y 370.096,Z 268.555,A -85,B 0,C 180,E1 -12733.127,E2 -12733.127} C_VEL
LIN {X 0,Y 369.706,Z 265.511,A -85,B 0,C 180,E1 -12736.249,E2 -12736.249} C_VEL
LIN {X 0,Y 369.266,Z 262.458,A -85,B 0,C 180,E1 -12739.671,E2 -12739.671} C_VEL
LIN {X 0,Y 368.923,Z 260.202,A -85,B 0,C 180,E1 -12742.434,E2 -12742.434} C_VEL
LIN {X 0,Y 368.94,Z 260.03,A -85,B 0,C 180,E1 -12745.142,E2 -12745.142} C_VEL
LIN {X 0,Y 368.905,Z 260.031,A -85,B 0,C 180,E1 -12749.039,E2 -12749.039} C_VEL
LIN {X 0,Y 368.915,Z 260.028,A -85,B 0,C 180,E1 -12751.553,E2 -12751.553} C_VEL
LIN {X 0,Y 368.926,Z 260.028,A -85,B 0,C 180,E1 -12754.009,E2 -12754.009} C_VEL
LIN {X 0,Y 368.902,Z 260.03,A -85,B 0,C 180,E1 -12757.598,E2 -12757.598} C_VEL
LIN {X 0,Y 368.917,Z 260.028,A -85,B 0,C 180,E1 -12761.098,E2 -12761.098} C_VEL
LIN {X 0,Y 368.942,Z 260.027,A -85,B 0,C 180,E1 -12764.527,E2 -12764.527} C_VEL
LIN {X 0,Y 369.059,Z 260.01,A -85,B 0,C 180,E1 -12766.785,E2 -12766.785} C_VEL
LIN {X 0,Y 369.061,Z 260.014,A -85,B 0,C 180,E1 -12770.126,E2 -12770.126} C_VEL
LIN {X 0,Y 369.151,Z 260,A -85,B 0,C 180,E1 -12773.435,E2 -12773.435} C_VEL
LIN {X 0,Y 369.295,Z 259.986,A -85,B 0,C 180,E1 -12777.812,E2 -12777.812} C_VEL
LIN {X 0,Y 369.299,Z 259.981,A -85,B 0,C 180,E1 -12782.175,E2 -12782.175} C_VEL
LIN {X 0,Y 369.167,Z 259.996,A -85,B 0,C 180,E1 -12786.552,E2 -12786.552} C_VEL
LIN {X 0,Y 369.048,Z 260.013,A -85,B 0,C 180,E1 -12789.862,E2 -12789.862} C_VEL
LIN {X 0,Y 369.02,Z 260.016,A -85,B 0,C 180,E1 -12793.765,E2 -12793.765} C_VEL
LIN {X 0,Y 368.97,Z 260.022,A -85,B 0,C 180,E1 -12797.736,E2 -12797.736} C_VEL
LIN {X 0,Y 368.886,Z 260.036,A -85,B 0,C 180,E1 -12801.214,E2 -12801.214} C_VEL
LIN {X 0,Y 368.928,Z 260.031,A -85,B 0,C 180,E1 -12804.769,E2 -12804.769} C_VEL
LIN {X 0,Y 368.934,Z 260.029,A -85,B 0,C 180,E1 -12807.197,E2 -12807.197} C_VEL
LIN {X 0,Y 368.897,Z 260.034,A -85,B 0,C 180,E1 -12810.947,E2 -12810.947} C_VEL
LIN {X 0,Y 368.893,Z 260.033,A -85,B 0,C 180,E1 -12814.995,E2 -12814.995} C_VEL
LIN {X 0,Y 368.867,Z 260.039,A -85,B 0,C 180,E1 -12818.634,E2 -12818.634} C_VEL
LIN {X 0,Y 368.899,Z 260.032,A -85,B 0,C 180,E1 -12822.014,E2 -12822.014} C_VEL
LIN {X 0,Y 368.946,Z 260.024,A -85,B 0,C 180,E1 -12825.187,E2 -12825.187} C_VEL
LIN {X 0,Y 368.895,Z 260.036,A -85,B 0,C 180,E1 -12828.18,E2 -12828.18} C_VEL
LIN {X 0,Y 368.863,Z 260.035,A -85,B 0,C 180,E1 -12831.354,E2 -12831.354} C_VEL
LIN {X 0,Y 368.885,Z 260.032,A -85,B 0,C 180,E1 -12835.142,E2 -12835.142} C_VEL
LIN {X 0,Y 368.876,Z 260.033,A -85,B 0,C 180,E1 -12839.042,E2 -12839.042} C_VEL
LIN {X 0,Y 368.931,Z 260.029,A -85,B 0,C 180,E1 -12841.56,E2 -12841.56} C_VEL
LIN {X 0,Y 368.905,Z 260.031,A -85,B 0,C 180,E1 -12845.221,E2 -12845.221} C_VEL
LIN {X 0,Y 368.933,Z 260.026,A -85,B 0,C 180,E1 -12848.949,E2 -12848.949} C_VEL
LIN {X 0,Y 368.932,Z 260.031,A -85,B 0,C 180,E1 -12852.255,E2 -12852.255} C_VEL
LIN {X 0,Y 368.984,Z 260.212,A -85,B 0,C 180,E1 -12855.418,E2 -12855.418} C_VEL
LIN {X 0,Y 369.813,Z 262.632,A -85,B 0,C 180,E1 -12855.706,E2 -12855.706} C_VEL
LIN {X 0,Y 371.642,Z 264.733,A -85,B 0,C 180,E1 -12856.274,E2 -12856.274} C_VEL
LIN {X 0,Y 373.74,Z 266.185,A -85,B 0,C 180,E1 -12856.912,E2 -12856.912} C_VEL
LIN {X 0,Y 375.395,Z 268.949,A -85,B 0,C 180,E1 -12857.498,E2 -12857.498} C_VEL
LIN {X 0,Y 377.651,Z 271.041,A -85,B 0,C 180,E1 -12858.296,E2 -12858.296} C_VEL
LIN {X 0,Y 379.318,Z 272.087,A -85,B 0,C 180,E1 -12858.887,E2 -12858.887} C_VEL
LIN {X 0,Y 381.079,Z 274.81,A -85,B 0,C 180,E1 -12859.641,E2 -12859.641} C_VEL
LIN {X 0,Y 383.643,Z 277.052,A -85,B 0,C 180,E1 -12860.754,E2 -12860.754} C_VEL
LIN {X 0,Y 386.027,Z 278.386,A -85,B 0,C 180,E1 -12861.879,E2 -12861.879} C_VEL
LIN {X 0,Y 387.956,Z 281.222,A -85,B 0,C 180,E1 -12863.046,E2 -12863.046} C_VEL
LIN {X 0,Y 389.984,Z 283.183,A -85,B 0,C 180,E1 -12864.441,E2 -12864.441} C_VEL
LIN {X 0,Y 391.641,Z 284.164,A -85,B 0,C 180,E1 -12865.884,E2 -12865.884} C_VEL
LIN {X 0,Y 393.217,Z 284.545,A -85,B 0,C 180,E1 -12867.951,E2 -12867.951} C_VEL
LIN {X 0,Y 393.777,Z 284.601,A -85,B 0,C 180,E1 -12870,E2 -12870} C_VEL
LIN {X 0,Y 393.217,Z 284.541,A -85,B 0,C 180,E1 -12872.049,E2 -12872.049} C_VEL
LIN {X 0,Y 391.641,Z 284.165,A -85,B 0,C 180,E1 -12874.116,E2 -12874.116} C_VEL
LIN {X 0,Y 389.612,Z 282.894,A -85,B 0,C 180,E1 -12875.823,E2 -12875.823} C_VEL
LIN {X 0,Y 387.673,Z 280.88,A -85,B 0,C 180,E1 -12877.137,E2 -12877.137} C_VEL
LIN {X 0,Y 385.889,Z 278.109,A -85,B 0,C 180,E1 -12878.208,E2 -12878.208} C_VEL
LIN {X 0,Y 382.912,Z 276.524,A -85,B 0,C 180,E1 -12879.575,E2 -12879.575} C_VEL
LIN {X 0,Y 380.56,Z 274.151,A -85,B 0,C 180,E1 -12880.575,E2 -12880.575} C_VEL
LIN {X 0,Y 379.096,Z 271.746,A -85,B 0,C 180,E1 -12881.204,E2 -12881.204} C_VEL
LIN {X 0,Y 376.435,Z 270.101,A -85,B 0,C 180,E1 -12882.125,E2 -12882.125} C_VEL
LIN {X 0,Y 374.304,Z 267.34,A -85,B 0,C 180,E1 -12882.889,E2 -12882.889} C_VEL
LIN {X 0,Y 373.42,Z 265.746,A -85,B 0,C 180,E1 -12883.192,E2 -12883.192} C_VEL
LIN {X 0,Y 370.867,Z 264.019,A -85,B 0,C 180,E1 -12883.969,E2 -12883.969} C_VEL
LIN {X 0,Y 369.4,Z 261.78,A -85,B 0,C 180,E1 -12884.425,E2 -12884.425} C_VEL
LIN {X 0,Y 368.962,Z 260.028,A -85,B 0,C 180,E1 -12884.618,E2 -12884.618} C_VEL
LIN {X 0,Y 368.942,Z 260.029,A -85,B 0,C 180,E1 -12887.771,E2 -12887.771} C_VEL
LIN {X 0,Y 368.929,Z 260.026,A -85,B 0,C 180,E1 -12891.219,E2 -12891.219} C_VEL
LIN {X 0,Y 368.905,Z 260.031,A -85,B 0,C 180,E1 -12894.779,E2 -12894.779} C_VEL
LIN {X 0,Y 368.931,Z 260.029,A -85,B 0,C 180,E1 -12898.44,E2 -12898.44} C_VEL
LIN {X 0,Y 368.856,Z 260.039,A -85,B 0,C 180,E1 -12902.241,E2 -12902.241} C_VEL
LIN {X 0,Y 368.877,Z 260.033,A -85,B 0,C 180,E1 -12905.006,E2 -12905.006} C_VEL
LIN {X 0,Y 368.863,Z 260.035,A -85,B 0,C 180,E1 -12908.646,E2 -12908.646} C_VEL
LIN {X 0,Y 368.896,Z 260.034,A -85,B 0,C 180,E1 -12912.025,E2 -12912.025} C_VEL
LIN {X 0,Y 368.94,Z 260.025,A -85,B 0,C 180,E1 -12914.737,E2 -12914.737} C_VEL
LIN {X 0,Y 368.322,Z 260.108,A -85,B 0,C 180,E1 -12915.648,E2 -12915.648} C_VEL
LIN {X 0,Y 365.471,Z 260.463,A -85,B 0,C 180,E1 -12917.128,E2 -12917.128} C_VEL
LIN {X 0,Y 363.013,Z 260.768,A -85,B 0,C 180,E1 -12918.325,E2 -12918.325} C_VEL
LIN {X 0,Y 361.94,Z 260.9,A -85,B 0,C 180,E1 -12919.252,E2 -12919.252} C_VEL
LIN {X 0,Y 361.845,Z 260.91,A -85,B 0,C 180,E1 -12919.566,E2 -12919.566} C_VEL
LIN {X 0,Y 361.828,Z 260.913,A -85,B 0,C 180,E1 -12922.988,E2 -12922.988} C_VEL
LIN {X 0,Y 361.824,Z 260.912,A -85,B 0,C 180,E1 -12926.637,E2 -12926.637} C_VEL
LIN {X 0,Y 361.841,Z 260.911,A -85,B 0,C 180,E1 -12929.679,E2 -12929.679} C_VEL
LIN {X 0,Y 361.925,Z 260.901,A -85,B 0,C 180,E1 -12933.482,E2 -12933.482} C_VEL
LIN {X 0,Y 361.857,Z 260.912,A -85,B 0,C 180,E1 -12937.151,E2 -12937.151} C_VEL
LIN {X 0,Y 361.879,Z 260.909,A -85,B 0,C 180,E1 -12940.73,E2 -12940.73} C_VEL
LIN {X 0,Y 361.923,Z 260.9,A -85,B 0,C 180,E1 -12944.233,E2 -12944.233} C_VEL
LIN {X 0,Y 361.982,Z 260.896,A -85,B 0,C 180,E1 -12946.535,E2 -12946.535} C_VEL
LIN {X 0,Y 361.985,Z 260.892,A -85,B 0,C 180,E1 -12949.944,E2 -12949.944} C_VEL
LIN {X 0,Y 362.13,Z 260.873,A -85,B 0,C 180,E1 -12953.32,E2 -12953.32} C_VEL
LIN {X 0,Y 362.262,Z 260.858,A -85,B 0,C 180,E1 -12957.783,E2 -12957.783} C_VEL
LIN {X 0,Y 362.257,Z 260.863,A -85,B 0,C 180,E1 -12962.23,E2 -12962.23} C_VEL
LIN {X 0,Y 362.115,Z 260.876,A -85,B 0,C 180,E1 -12966.693,E2 -12966.693} C_VEL
LIN {X 0,Y 361.998,Z 260.895,A -85,B 0,C 180,E1 -12970.069,E2 -12970.069} C_VEL
LIN {X 0,Y 361.982,Z 260.898,A -85,B 0,C 180,E1 -12973.892,E2 -12973.892} C_VEL
LIN {X 0,Y 361.89,Z 260.906,A -85,B 0,C 180,E1 -12978.109,E2 -12978.109} C_VEL
LIN {X 0,Y 361.859,Z 260.913,A -85,B 0,C 180,E1 -12981.661,E2 -12981.661} C_VEL
LIN {X 0,Y 361.859,Z 260.91,A -85,B 0,C 180,E1 -12985.301,E2 -12985.301} C_VEL
LIN {X 0,Y 361.864,Z 260.909,A -85,B 0,C 180,E1 -12989.078,E2 -12989.078} C_VEL
LIN {X 0,Y 361.857,Z 260.91,A -85,B 0,C 180,E1 -12992.949,E2 -12992.949} C_VEL
LIN {X 0,Y 361.874,Z 260.909,A -85,B 0,C 180,E1 -12995.641,E2 -12995.641} C_VEL
LIN {X 0,Y 361.9,Z 261.117,A -85,B 0,C 180,E1 -12997.232,E2 -12997.232} C_VEL
LIN {X 0,Y 362.282,Z 264.039,A -85,B 0,C 180,E1 -13000.838,E2 -13000.838} C_VEL
LIN {X 0,Y 362.749,Z 267.045,A -85,B 0,C 180,E1 -13004.23,E2 -13004.23} C_VEL
LIN {X 0,Y 363.049,Z 270.112,A -85,B 0,C 180,E1 -13007.365,E2 -13007.365} C_VEL
LIN {X 0,Y 362.887,Z 273.203,A -85,B 0,C 180,E1 -13010.276,E2 -13010.276} C_VEL
LIN {X 0,Y 362.54,Z 276.367,A -85,B 0,C 180,E1 -13013.063,E2 -13013.063} C_VEL
LIN {X 0,Y 362.052,Z 280.607,A -85,B 0,C 180,E1 -13016.591,E2 -13016.591} C_VEL
LIN {X 0,Y 361.666,Z 284.465,A -85,B 0,C 180,E1 -13019.653,E2 -13019.653} C_VEL
LIN {X 0,Y 361.251,Z 289.543,A -85,B 0,C 180,E1 -13023.505,E2 -13023.505} C_VEL
LIN {X 0,Y 360.875,Z 294.435,A -85,B 0,C 180,E1 -13027.077,E2 -13027.077} C_VEL
LIN {X 0,Y 360.73,Z 298.552,A -85,B 0,C 180,E1 -13029.945,E2 -13029.945} C_VEL
LIN {X 0,Y 362.949,Z 308.991,A -85,B 0,C 180,E1 -13030.438,E2 -13030.438} C_VEL
LIN {X 0,Y 364.676,Z 318.469,A -85,B 0,C 180,E1 -13030.999,E2 -13030.999} C_VEL
LIN {X 0,Y 366.071,Z 328.221,A -85,B 0,C 180,E1 -13031.693,E2 -13031.693} C_VEL
LIN {X 0,Y 366.744,Z 333.912,A -85,B 0,C 180,E1 -13032.145,E2 -13032.145} C_VEL
LIN {X 0,Y 365.724,Z 344.824,A -85,B 0,C 180,E1 -13033.103,E2 -13033.103} C_VEL
LIN {X 0,Y 364.829,Z 353.771,A -85,B 0,C 180,E1 -13034.068,E2 -13034.068} C_VEL
LIN {X 0,Y 364.147,Z 360.931,A -85,B 0,C 180,E1 -13034.979,E2 -13034.979} C_VEL
LIN {X 0,Y 363.289,Z 369.53,A -85,B 0,C 180,E1 -13036.292,E2 -13036.292} C_VEL
LIN {X 0,Y 362.583,Z 375.734,A -85,B 0,C 180,E1 -13037.405,E2 -13037.405} C_VEL
LIN {X 0,Y 361.802,Z 382.272,A -85,B 0,C 180,E1 -13038.799,E2 -13038.799} C_VEL
LIN {X 0,Y 361.383,Z 386.777,A -85,B 0,C 180,E1 -13039.92,E2 -13039.92} C_VEL
LIN {X 0,Y 360.866,Z 392.271,A -85,B 0,C 180,E1 -13041.601,E2 -13041.601} C_VEL
LIN {X 0,Y 360.537,Z 396.598,A -85,B 0,C 180,E1 -13043.284,E2 -13043.284} C_VEL
LIN {X 0,Y 360.423,Z 398.967,A -85,B 0,C 180,E1 -13044.405,E2 -13044.405} C_VEL
LIN {X 0,Y 360.388,Z 400.768,A -85,B 0,C 180,E1 -13045.526,E2 -13045.526} C_VEL
LIN {X 0,Y 360.27,Z 403.213,A -85,B 0,C 180,E1 -13047.764,E2 -13047.764} C_VEL
LIN {X 0,Y 360.3,Z 403.803,A -85,B 0,C 180,E1 -13048.882,E2 -13048.882} C_VEL
LIN {X 0,Y 360.3,Z 403.803,A -85,B 0,C 180,E1 -13051.118,E2 -13051.118} C_VEL
LIN {X 0,Y 360.27,Z 403.213,A -85,B 0,C 180,E1 -13052.236,E2 -13052.236} C_VEL
LIN {X 0,Y 360.388,Z 400.768,A -85,B 0,C 180,E1 -13054.474,E2 -13054.474} C_VEL
LIN {X 0,Y 360.462,Z 398.02,A -85,B 0,C 180,E1 -13056.062,E2 -13056.062} C_VEL
LIN {X 0,Y 360.743,Z 393.826,A -85,B 0,C 180,E1 -13057.838,E2 -13057.838} C_VEL
LIN {X 0,Y 361.19,Z 388.694,A -85,B 0,C 180,E1 -13059.52,E2 -13059.52} C_VEL
LIN {X 0,Y 361.708,Z 383.429,A -85,B 0,C 180,E1 -13060.92,E2 -13060.92} C_VEL
LIN {X 0,Y 362.401,Z 377.11,A -85,B 0,C 180,E1 -13062.317,E2 -13062.317} C_VEL
LIN {X 0,Y 363.067,Z 371.157,A -85,B 0,C 180,E1 -13063.432,E2 -13063.432} C_VEL
LIN {X 0,Y 363.782,Z 364.226,A -85,B 0,C 180,E1 -13064.545,E2 -13064.545} C_VEL
LIN {X 0,Y 364.564,Z 356.041,A -85,B 0,C 180,E1 -13065.657,E2 -13065.657} C_VEL
LIN {X 0,Y 365.448,Z 347.528,A -85,B 0,C 180,E1 -13066.622,E2 -13066.622} C_VEL
LIN {X 0,Y 366.302,Z 338.81,A -85,B 0,C 180,E1 -13067.444,E2 -13067.444} C_VEL
LIN {X 0,Y 366.616,Z 332.878,A -85,B 0,C 180,E1 -13067.945,E2 -13067.945} C_VEL
LIN {X 0,Y 365.015,Z 320.597,A -85,B 0,C 180,E1 -13068.863,E2 -13068.863} C_VEL
LIN {X 0,Y 363.068,Z 309.685,A -85,B 0,C 180,E1 -13069.526,E2 -13069.526} C_VEL
LIN {X 0,Y 360.836,Z 299.404,A -85,B 0,C 180,E1 -13070.025,E2 -13070.025} C_VEL
LIN {X 0,Y 360.721,Z 298.389,A -85,B 0,C 180,E1 -13070.083,E2 -13070.083} C_VEL
LIN {X 0,Y 361.003,Z 292.746,A -85,B 0,C 180,E1 -13074.131,E2 -13074.131} C_VEL
LIN {X 0,Y 361.395,Z 287.759,A -85,B 0,C 180,E1 -13077.821,E2 -13077.821} C_VEL
LIN {X 0,Y 361.829,Z 282.824,A -85,B 0,C 180,E1 -13081.63,E2 -13081.63} C_VEL
LIN {X 0,Y 362.343,Z 278.14,A -85,B 0,C 180,E1 -13085.443,E2 -13085.443} C_VEL
LIN {X 0,Y 362.741,Z 274.775,A -85,B 0,C 180,E1 -13088.315,E2 -13088.315} C_VEL
LIN {X 0,Y 363.033,Z 271.624,A -85,B 0,C 180,E1 -13091.163,E2 -13091.163} C_VEL
LIN {X 0,Y 363.098,Z 270.063,A -85,B 0,C 180,E1 -13092.644,E2 -13092.644} C_VEL
LIN {X 0,Y 362.747,Z 267.018,A -85,B 0,C 180,E1 -13095.794,E2 -13095.794} C_VEL
LIN {X 0,Y 362.299,Z 264.02,A -85,B 0,C 180,E1 -13099.158,E2 -13099.158} C_VEL
LIN {X 0,Y 361.877,Z 260.963,A -85,B 0,C 180,E1 -13102.978,E2 -13102.978} C_VEL
LIN {X 0,Y 361.867,Z 260.912,A -85,B 0,C 180,E1 -13106.627,E2 -13106.627} C_VEL
LIN {X 0,Y 361.856,Z 260.907,A -85,B 0,C 180,E1 -13109.665,E2 -13109.665} C_VEL
LIN {X 0,Y 361.862,Z 260.907,A -85,B 0,C 180,E1 -13113.462,E2 -13113.462} C_VEL
LIN {X 0,Y 361.867,Z 260.906,A -85,B 0,C 180,E1 -13117.138,E2 -13117.138} C_VEL
LIN {X 0,Y 361.857,Z 260.909,A -85,B 0,C 180,E1 -13120.715,E2 -13120.715} C_VEL
LIN {X 0,Y 361.897,Z 260.908,A -85,B 0,C 180,E1 -13124.218,E2 -13124.218} C_VEL
LIN {X 0,Y 362.001,Z 260.891,A -85,B 0,C 180,E1 -13126.522,E2 -13126.522} C_VEL
LIN {X 0,Y 361.998,Z 260.895,A -85,B 0,C 180,E1 -13129.931,E2 -13129.931} C_VEL
LIN {X 0,Y 362.115,Z 260.876,A -85,B 0,C 180,E1 -13133.307,E2 -13133.307} C_VEL
LIN {X 0,Y 362.258,Z 260.863,A -85,B 0,C 180,E1 -13137.77,E2 -13137.77} C_VEL
LIN {X 0,Y 362.262,Z 260.858,A -85,B 0,C 180,E1 -13142.217,E2 -13142.217} C_VEL
LIN {X 0,Y 362.13,Z 260.873,A -85,B 0,C 180,E1 -13146.68,E2 -13146.68} C_VEL
LIN {X 0,Y 361.985,Z 260.892,A -85,B 0,C 180,E1 -13150.056,E2 -13150.056} C_VEL
LIN {X 0,Y 361.981,Z 260.893,A -85,B 0,C 180,E1 -13153.892,E2 -13153.892} C_VEL
LIN {X 0,Y 361.907,Z 260.904,A -85,B 0,C 180,E1 -13156.927,E2 -13156.927} C_VEL
LIN {X 0,Y 361.86,Z 260.908,A -85,B 0,C 180,E1 -13160.454,E2 -13160.454} C_VEL
LIN {X 0,Y 361.867,Z 260.906,A -85,B 0,C 180,E1 -13164.106,E2 -13164.106} C_VEL
LIN {X 0,Y 361.913,Z 260.905,A -85,B 0,C 180,E1 -13166.714,E2 -13166.714} C_VEL
LIN {X 0,Y 361.841,Z 260.911,A -85,B 0,C 180,E1 -13170.321,E2 -13170.321} C_VEL
LIN {X 0,Y 361.819,Z 260.914,A -85,B 0,C 180,E1 -13174.274,E2 -13174.274} C_VEL
LIN {X 0,Y 361.824,Z 260.912,A -85,B 0,C 180,E1 -13177.216,E2 -13177.216} C_VEL
LIN {X 0,Y 361.865,Z 260.909,A -85,B 0,C 180,E1 -13180.762,E2 -13180.762} C_VEL
LIN {X 0,Y 361.889,Z 260.909,A -85,B 0,C 180,E1 -13184.345,E2 -13184.345} C_VEL
LIN {X 0,Y 361.841,Z 260.91,A -85,B 0,C 180,E1 -13187.554,E2 -13187.554} C_VEL
LIN {X 0,Y 361.826,Z 260.911,A -85,B 0,C 180,E1 -13190.967,E2 -13190.967} C_VEL
LIN {X 0,Y 361.823,Z 260.912,A -85,B 0,C 180,E1 -13194.65,E2 -13194.65} C_VEL
LIN {X 0,Y 361.806,Z 260.916,A -85,B 0,C 180,E1 -13198.368,E2 -13198.368} C_VEL
LIN {X 0,Y 361.867,Z 260.908,A -85,B 0,C 180,E1 -13202.218,E2 -13202.218} C_VEL
LIN {X 0,Y 361.876,Z 260.909,A -85,B 0,C 180,E1 -13205.87,E2 -13205.87} C_VEL
LIN {X 0,Y 361.871,Z 260.911,A -85,B 0,C 180,E1 -13209.539,E2 -13209.539} C_VEL
LIN {X 0,Y 361.875,Z 260.91,A -85,B 0,C 180,E1 -13213.064,E2 -13213.064} C_VEL
LIN {X 0,Y 361.879,Z 260.909,A -85,B 0,C 180,E1 -13213.753,E2 -13213.753} C_VEL
LIN {X 0,Y 362.828,Z 263.671,A -85,B 0,C 180,E1 -13214.074,E2 -13214.074} C_VEL
LIN {X 0,Y 364.898,Z 265.865,A -85,B 0,C 180,E1 -13214.615,E2 -13214.615} C_VEL
LIN {X 0,Y 366.26,Z 266.855,A -85,B 0,C 180,E1 -13214.977,E2 -13214.977} C_VEL
LIN {X 0,Y 368.171,Z 269.927,A -85,B 0,C 180,E1 -13215.561,E2 -13215.561} C_VEL
LIN {X 0,Y 371,Z 272.175,A -85,B 0,C 180,E1 -13216.384,E2 -13216.384} C_VEL
LIN {X 0,Y 372.054,Z 273.665,A -85,B 0,C 180,E1 -13216.735,E2 -13216.735} C_VEL
LIN {X 0,Y 374.641,Z 276.716,A -85,B 0,C 180,E1 -13217.593,E2 -13217.593} C_VEL
LIN {X 0,Y 377.554,Z 278.865,A -85,B 0,C 180,E1 -13218.598,E2 -13218.598} C_VEL
LIN {X 0,Y 379.86,Z 281.898,A -85,B 0,C 180,E1 -13219.54,E2 -13219.54} C_VEL
LIN {X 0,Y 382.671,Z 284.142,A -85,B 0,C 180,E1 -13220.73,E2 -13220.73} C_VEL
LIN {X 0,Y 384.645,Z 285.238,A -85,B 0,C 180,E1 -13221.637,E2 -13221.637} C_VEL
LIN {X 0,Y 386.76,Z 288.125,A -85,B 0,C 180,E1 -13222.868,E2 -13222.868} C_VEL
LIN {X 0,Y 388.89,Z 290.129,A -85,B 0,C 180,E1 -13224.296,E2 -13224.296} C_VEL
LIN {X 0,Y 390.753,Z 291.192,A -85,B 0,C 180,E1 -13225.874,E2 -13225.874} C_VEL
LIN {X 0,Y 392.355,Z 291.587,A -85,B 0,C 180,E1 -13227.947,E2 -13227.947} C_VEL
LIN {X 0,Y 392.773,Z 291.626,A -85,B 0,C 180,E1 -13228.975,E2 -13228.975} C_VEL
LIN {X 0,Y 392.912,Z 291.647,A -85,B 0,C 180,E1 -13230,E2 -13230} C_VEL
LIN {X 0,Y 392.773,Z 291.629,A -85,B 0,C 180,E1 -13231.025,E2 -13231.025} C_VEL
LIN {X 0,Y 391.687,Z 291.421,A -85,B 0,C 180,E1 -13233.086,E2 -13233.086} C_VEL
LIN {X 0,Y 389.884,Z 290.783,A -85,B 0,C 180,E1 -13234.912,E2 -13234.912} C_VEL
LIN {X 0,Y 387.664,Z 289.107,A -85,B 0,C 180,E1 -13236.555,E2 -13236.555} C_VEL
LIN {X 0,Y 385.324,Z 286.321,A -85,B 0,C 180,E1 -13237.967,E2 -13237.967} C_VEL
LIN {X 0,Y 384.271,Z 284.89,A -85,B 0,C 180,E1 -13238.546,E2 -13238.546} C_VEL
LIN {X 0,Y 381.217,Z 283.123,A -85,B 0,C 180,E1 -13239.906,E2 -13239.906} C_VEL
LIN {X 0,Y 378.415,Z 280.193,A -85,B 0,C 180,E1 -13241.049,E2 -13241.049} C_VEL
LIN {X 0,Y 377.3,Z 278.492,A -85,B 0,C 180,E1 -13241.498,E2 -13241.498} C_VEL
LIN {X 0,Y 374.296,Z 276.378,A -85,B 0,C 180,E1 -13242.522,E2 -13242.522} C_VEL
LIN {X 0,Y 371.82,Z 273.31,A -85,B 0,C 180,E1 -13243.343,E2 -13243.343} C_VEL
LIN {X 0,Y 371,Z 272.175,A -85,B 0,C 180,E1 -13243.616,E2 -13243.616} C_VEL
LIN {X 0,Y 368.225,Z 269.964,A -85,B 0,C 180,E1 -13244.424,E2 -13244.424} C_VEL
LIN {X 0,Y 366.296,Z 266.964,A -85,B 0,C 180,E1 -13245.01,E2 -13245.01} C_VEL
LIN {X 0,Y 365.806,Z 266.378,A -85,B 0,C 180,E1 -13245.153,E2 -13245.153} C_VEL
LIN {X 0,Y 363.429,Z 264.52,A -85,B 0,C 180,E1 -13245.762,E2 -13245.762} C_VEL
LIN {X 0,Y 362.164,Z 262.176,A -85,B 0,C 180,E1 -13246.125,E2 -13246.125} C_VEL
LIN {X 0,Y 361.868,Z 260.911,A -85,B 0,C 180,E1 -13246.284,E2 -13246.284} C_VEL
LIN {X 0,Y 361.876,Z 260.909,A -85,B 0,C 180,E1 -13249.278,E2 -13249.278} C_VEL
LIN {X 0,Y 361.865,Z 260.908,A -85,B 0,C 180,E1 -13252.857,E2 -13252.857} C_VEL
LIN {X 0,Y 361.887,Z 260.905,A -85,B 0,C 180,E1 -13256.725,E2 -13256.725} C_VEL
LIN {X 0,Y 361.823,Z 260.915,A -85,B 0,C 180,E1 -13260.332,E2 -13260.332} C_VEL
LIN {X 0,Y 361.804,Z 260.917,A -85,B 0,C 180,E1 -13264.285,E2 -13264.285} C_VEL
LIN {X 0,Y 361.815,Z 260.913,A -85,B 0,C 180,E1 -13267.228,E2 -13267.228} C_VEL
LIN {X 0,Y 361.859,Z 260.907,A -85,B 0,C 180,E1 -13270.774,E2 -13270.774} C_VEL
LIN {X 0,Y 361.87,Z 260.905,A -85,B 0,C 180,E1 -13274.732,E2 -13274.732} C_VEL
LIN {X 0,Y 361.844,Z 260.915,A -85,B 0,C 180,E1 -13277.566,E2 -13277.566} C_VEL
LIN {X 0,Y 361.845,Z 260.91,A -85,B 0,C 180,E1 -13279.566,E2 -13279.566} C_VEL
LIN {X 0,Y 361.161,Z 260.994,A -85,B 0,C 180,E1 -13280.495,E2 -13280.495} C_VEL
LIN {X 0,Y 358.312,Z 261.35,A -85,B 0,C 180,E1 -13282.005,E2 -13282.005} C_VEL
LIN {X 0,Y 355.906,Z 261.653,A -85,B 0,C 180,E1 -13283.226,E2 -13283.226} C_VEL
LIN {X 0,Y 354.867,Z 261.778,A -85,B 0,C 180,E1 -13284.171,E2 -13284.171} C_VEL
LIN {X 0,Y 354.778,Z 261.789,A -85,B 0,C 180,E1 -13284.491,E2 -13284.491} C_VEL
LIN {X 0,Y 354.753,Z 261.794,A -85,B 0,C 180,E1 -13287.673,E2 -13287.673} C_VEL
LIN {X 0,Y 354.817,Z 261.786,A -85,B 0,C 180,E1 -13291.625,E2 -13291.625} C_VEL
LIN {X 0,Y 354.871,Z 261.777,A -85,B 0,C 180,E1 -13294.179,E2 -13294.179} C_VEL
LIN {X 0,Y 354.792,Z 261.787,A -85,B 0,C 180,E1 -13297.9,E2 -13297.9} C_VEL
LIN {X 0,Y 354.869,Z 261.778,A -85,B 0,C 180,E1 -13301.915,E2 -13301.915} C_VEL
LIN {X 0,Y 354.925,Z 261.771,A -85,B 0,C 180,E1 -13305.989,E2 -13305.989} C_VEL
LIN {X 0,Y 354.941,Z 261.769,A -85,B 0,C 180,E1 -13309.742,E2 -13309.742} C_VEL
LIN {X 0,Y 355.094,Z 261.75,A -85,B 0,C 180,E1 -13313.187,E2 -13313.187} C_VEL
LIN {X 0,Y 355.225,Z 261.734,A -85,B 0,C 180,E1 -13317.739,E2 -13317.739} C_VEL
LIN {X 0,Y 355.165,Z 261.741,A -85,B 0,C 180,E1 -13321.14,E2 -13321.14} C_VEL
LIN {X 0,Y 355.22,Z 261.74,A -85,B 0,C 180,E1 -13322.274,E2 -13322.274} C_VEL
LIN {X 0,Y 355.082,Z 261.752,A -85,B 0,C 180,E1 -13326.827,E2 -13326.827} C_VEL
LIN {X 0,Y 354.955,Z 261.77,A -85,B 0,C 180,E1 -13330.271,E2 -13330.271} C_VEL
LIN {X 0,Y 354.925,Z 261.776,A -85,B 0,C 180,E1 -13334.011,E2 -13334.011} C_VEL
LIN {X 0,Y 354.848,Z 261.783,A -85,B 0,C 180,E1 -13338.074,E2 -13338.074} C_VEL
LIN {X 0,Y 354.812,Z 261.787,A -85,B 0,C 180,E1 -13342.113,E2 -13342.113} C_VEL
LIN {X 0,Y 354.802,Z 261.789,A -85,B 0,C 180,E1 -13345.841,E2 -13345.841} C_VEL
LIN {X 0,Y 354.802,Z 261.79,A -85,B 0,C 180,E1 -13349.689,E2 -13349.689} C_VEL
LIN {X 0,Y 354.796,Z 261.787,A -85,B 0,C 180,E1 -13352.338,E2 -13352.338} C_VEL
LIN {X 0,Y 354.829,Z 261.787,A -85,B 0,C 180,E1 -13355.702,E2 -13355.702} C_VEL
LIN {X 0,Y 354.803,Z 261.792,A -85,B 0,C 180,E1 -13356.464,E2 -13356.464} C_VEL
LIN {X 0,Y 355.135,Z 264.044,A -85,B 0,C 180,E1 -13359.486,E2 -13359.486} C_VEL
LIN {X 0,Y 355.561,Z 267.008,A -85,B 0,C 180,E1 -13363.002,E2 -13363.002} C_VEL
LIN {X 0,Y 355.925,Z 270.048,A -85,B 0,C 180,E1 -13366.284,E2 -13366.284} C_VEL
LIN {X 0,Y 355.932,Z 273.156,A -85,B 0,C 180,E1 -13369.339,E2 -13369.339} C_VEL
LIN {X 0,Y 355.629,Z 276.317,A -85,B 0,C 180,E1 -13372.237,E2 -13372.237} C_VEL
LIN {X 0,Y 355.22,Z 279.483,A -85,B 0,C 180,E1 -13374.988,E2 -13374.988} C_VEL
LIN {X 0,Y 354.697,Z 284.346,A -85,B 0,C 180,E1 -13378.992,E2 -13378.992} C_VEL
LIN {X 0,Y 354.371,Z 287.617,A -85,B 0,C 180,E1 -13381.578,E2 -13381.578} C_VEL
LIN {X 0,Y 354.083,Z 290.922,A -85,B 0,C 180,E1 -13384.109,E2 -13384.109} C_VEL
LIN {X 0,Y 353.838,Z 294.266,A -85,B 0,C 180,E1 -13386.594,E2 -13386.594} C_VEL
LIN {X 0,Y 353.677,Z 298.196,A -85,B 0,C 180,E1 -13389.518,E2 -13389.518} C_VEL
LIN {X 0,Y 356.044,Z 309.493,A -85,B 0,C 180,E1 -13390.074,E2 -13390.074} C_VEL
LIN {X 0,Y 357.876,Z 319.507,A -85,B 0,C 180,E1 -13390.696,E2 -13390.696} C_VEL
LIN {X 0,Y 359.397,Z 330.646,A -85,B 0,C 180,E1 -13391.533,E2 -13391.533} C_VEL
LIN {X 0,Y 359.848,Z 335.335,A -85,B 0,C 180,E1 -13391.938,E2 -13391.938} C_VEL
LIN {X 0,Y 358.935,Z 344.612,A -85,B 0,C 180,E1 -13392.774,E2 -13392.774} C_VEL
LIN {X 0,Y 357.976,Z 353.559,A -85,B 0,C 180,E1 -13393.754,E2 -13393.754} C_VEL
LIN {X 0,Y 357.187,Z 361.453,A -85,B 0,C 180,E1 -13394.791,E2 -13394.791} C_VEL
LIN {X 0,Y 356.359,Z 369.318,A -85,B 0,C 180,E1 -13396.02,E2 -13396.02} C_VEL
LIN {X 0,Y 355.621,Z 375.522,A -85,B 0,C 180,E1 -13397.154,E2 -13397.154} C_VEL
LIN {X 0,Y 354.797,Z 382.06,A -85,B 0,C 180,E1 -13398.575,E2 -13398.575} C_VEL
LIN {X 0,Y 354.361,Z 386.565,A -85,B 0,C 180,E1 -13399.718,E2 -13399.718} C_VEL
LIN {X 0,Y 353.829,Z 392.06,A -85,B 0,C 180,E1 -13401.433,E2 -13401.433} C_VEL
LIN {X 0,Y 353.458,Z 396.386,A -85,B 0,C 180,E1 -13403.148,E2 -13403.148} C_VEL
LIN {X 0,Y 353.348,Z 398.755,A -85,B 0,C 180,E1 -13404.293,E2 -13404.293} C_VEL
LIN {X 0,Y 353.302,Z 400.557,A -85,B 0,C 180,E1 -13405.436,E2 -13405.436} C_VEL
LIN {X 0,Y 353.179,Z 403.002,A -85,B 0,C 180,E1 -13407.719,E2 -13407.719} C_VEL
LIN {X 0,Y 353.201,Z 403.592,A -85,B 0,C 180,E1 -13408.86,E2 -13408.86} C_VEL
LIN {X 0,Y 353.201,Z 403.592,A -85,B 0,C 180,E1 -13411.14,E2 -13411.14} C_VEL
LIN {X 0,Y 353.179,Z 403.002,A -85,B 0,C 180,E1 -13412.281,E2 -13412.281} C_VEL
LIN {X 0,Y 353.302,Z 400.557,A -85,B 0,C 180,E1 -13414.564,E2 -13414.564} C_VEL
LIN {X 0,Y 353.356,Z 398.197,A -85,B 0,C 180,E1 -13416.001,E2 -13416.001} C_VEL
LIN {X 0,Y 353.563,Z 395.145,A -85,B 0,C 180,E1 -13417.423,E2 -13417.423} C_VEL
LIN {X 0,Y 353.99,Z 390.399,A -85,B 0,C 180,E1 -13419.139,E2 -13419.139} C_VEL
LIN {X 0,Y 354.608,Z 384.374,A -85,B 0,C 180,E1 -13420.852,E2 -13420.852} C_VEL
LIN {X 0,Y 355.252,Z 378.274,A -85,B 0,C 180,E1 -13422.279,E2 -13422.279} C_VEL
LIN {X 0,Y 355.955,Z 372.572,A -85,B 0,C 180,E1 -13423.414,E2 -13423.414} C_VEL
LIN {X 0,Y 356.897,Z 364.014,A -85,B 0,C 180,E1 -13424.832,E2 -13424.832} C_VEL
LIN {X 0,Y 357.716,Z 355.829,A -85,B 0,C 180,E1 -13425.965,E2 -13425.965} C_VEL
LIN {X 0,Y 358.65,Z 347.316,A -85,B 0,C 180,E1 -13426.947,E2 -13426.947} C_VEL
LIN {X 0,Y 359.528,Z 338.599,A -85,B 0,C 180,E1 -13427.784,E2 -13427.784} C_VEL
LIN {X 0,Y 359.726,Z 333.692,A -85,B 0,C 180,E1 -13428.215,E2 -13428.215} C_VEL
LIN {X 0,Y 358.257,Z 321.864,A -85,B 0,C 180,E1 -13429.147,E2 -13429.147} C_VEL
LIN {X 0,Y 356.125,Z 309.628,A -85,B 0,C 180,E1 -13429.916,E2 -13429.916} C_VEL
LIN {X 0,Y 353.712,Z 298.843,A -85,B 0,C 180,E1 -13430.456,E2 -13430.456} C_VEL
LIN {X 0,Y 353.67,Z 298.169,A -85,B 0,C 180,E1 -13430.501,E2 -13430.501} C_VEL
LIN {X 0,Y 353.959,Z 292.583,A -85,B 0,C 180,E1 -13434.643,E2 -13434.643} C_VEL
LIN {X 0,Y 354.246,Z 289.266,A -85,B 0,C 180,E1 -13437.148,E2 -13437.148} C_VEL
LIN {X 0,Y 354.513,Z 285.982,A -85,B 0,C 180,E1 -13439.709,E2 -13439.709} C_VEL
LIN {X 0,Y 354.851,Z 282.717,A -85,B 0,C 180,E1 -13442.326,E2 -13442.326} C_VEL
LIN {X 0,Y 355.345,Z 278.548,A -85,B 0,C 180,E1 -13445.81,E2 -13445.81} C_VEL
LIN {X 0,Y 355.81,Z 274.711,A -85,B 0,C 180,E1 -13449.202,E2 -13449.202} C_VEL
LIN {X 0,Y 356.017,Z 271.575,A -85,B 0,C 180,E1 -13452.157,E2 -13452.157} C_VEL
LIN {X 0,Y 355.858,Z 269.107,A -85,B 0,C 180,E1 -13454.68,E2 -13454.68} C_VEL
LIN {X 0,Y 355.442,Z 266.345,A -85,B 0,C 180,E1 -13457.752,E2 -13457.752} C_VEL
LIN {X 0,Y 355.097,Z 263.897,A -85,B 0,C 180,E1 -13460.698,E2 -13460.698} C_VEL
LIN {X 0,Y 354.802,Z 261.789,A -85,B 0,C 180,E1 -13463.535,E2 -13463.535} C_VEL
LIN {X 0,Y 354.809,Z 261.79,A -85,B 0,C 180,E1 -13466.31,E2 -13466.31} C_VEL
LIN {X 0,Y 354.801,Z 261.789,A -85,B 0,C 180,E1 -13468.996,E2 -13468.996} C_VEL
LIN {X 0,Y 354.797,Z 261.787,A -85,B 0,C 180,E1 -13471.609,E2 -13471.609} C_VEL
LIN {X 0,Y 354.809,Z 261.785,A -85,B 0,C 180,E1 -13475.414,E2 -13475.414} C_VEL
LIN {X 0,Y 354.826,Z 261.783,A -85,B 0,C 180,E1 -13479.107,E2 -13479.107} C_VEL
LIN {X 0,Y 354.855,Z 261.781,A -85,B 0,C 180,E1 -13482.712,E2 -13482.712} C_VEL
LIN {X 0,Y 354.941,Z 261.773,A -85,B 0,C 180,E1 -13486.249,E2 -13486.249} C_VEL
LIN {X 0,Y 354.955,Z 261.77,A -85,B 0,C 180,E1 -13489.729,E2 -13489.729} C_VEL
LIN {X 0,Y 355.082,Z 261.752,A -85,B 0,C 180,E1 -13493.173,E2 -13493.173} C_VEL
LIN {X 0,Y 355.22,Z 261.74,A -85,B 0,C 180,E1 -13497.726,E2 -13497.726} C_VEL
LIN {X 0,Y 355.137,Z 261.745,A -85,B 0,C 180,E1 -13501.127,E2 -13501.127} C_VEL
LIN {X 0,Y 355.225,Z 261.734,A -85,B 0,C 180,E1 -13502.261,E2 -13502.261} C_VEL
LIN {X 0,Y 355.094,Z 261.75,A -85,B 0,C 180,E1 -13506.813,E2 -13506.813} C_VEL
LIN {X 0,Y 354.941,Z 261.769,A -85,B 0,C 180,E1 -13510.258,E2 -13510.258} C_VEL
LIN {X 0,Y 354.925,Z 261.771,A -85,B 0,C 180,E1 -13514.011,E2 -13514.011} C_VEL
LIN {X 0,Y 354.869,Z 261.778,A -85,B 0,C 180,E1 -13518.085,E2 -13518.085} C_VEL
LIN {X 0,Y 354.792,Z 261.787,A -85,B 0,C 180,E1 -13522.1,E2 -13522.1} C_VEL
LIN {X 0,Y 354.871,Z 261.777,A -85,B 0,C 180,E1 -13525.821,E2 -13525.821} C_VEL
LIN {X 0,Y 354.787,Z 261.788,A -85,B 0,C 180,E1 -13529.675,E2 -13529.675} C_VEL
LIN {X 0,Y 354.772,Z 261.79,A -85,B 0,C 180,E1 -13533.695,E2 -13533.695} C_VEL
LIN {X 0,Y 354.76,Z 261.796,A -85,B 0,C 180,E1 -13536.453,E2 -13536.453} C_VEL
LIN {X 0,Y 354.786,Z 261.788,A -85,B 0,C 180,E1 -13539.417,E2 -13539.417} C_VEL
LIN {X 0,Y 354.799,Z 261.788,A -85,B 0,C 180,E1 -13542.87,E2 -13542.87} C_VEL
LIN {X 0,Y 354.823,Z 261.788,A -85,B 0,C 180,E1 -13546.113,E2 -13546.113} C_VEL
LIN {X 0,Y 354.81,Z 261.785,A -85,B 0,C 180,E1 -13549.183,E2 -13549.183} C_VEL
LIN {X 0,Y 354.759,Z 261.795,A -85,B 0,C 180,E1 -13552.397,E2 -13552.397} C_VEL
LIN {X 0,Y 354.761,Z 261.791,A -85,B 0,C 180,E1 -13554.936,E2 -13554.936} C_VEL
LIN {X 0,Y 354.761,Z 261.793,A -85,B 0,C 180,E1 -13558.395,E2 -13558.395} C_VEL
LIN {X 0,Y 354.799,Z 261.79,A -85,B 0,C 180,E1 -13561.615,E2 -13561.615} C_VEL
LIN {X 0,Y 354.844,Z 261.783,A -85,B 0,C 180,E1 -13564.169,E2 -13564.169} C_VEL
LIN {X 0,Y 354.834,Z 261.786,A -85,B 0,C 180,E1 -13567.894,E2 -13567.894} C_VEL
LIN {X 0,Y 354.865,Z 261.783,A -85,B 0,C 180,E1 -13571.888,E2 -13571.888} C_VEL
LIN {X 0,Y 354.879,Z 261.944,A -85,B 0,C 180,E1 -13572.331,E2 -13572.331} C_VEL
LIN {X 0,Y 355.709,Z 264.398,A -85,B 0,C 180,E1 -13572.58,E2 -13572.58} C_VEL
LIN {X 0,Y 357.601,Z 266.578,A -85,B 0,C 180,E1 -13573.036,E2 -13573.036} C_VEL
LIN {X 0,Y 358.839,Z 267.55,A -85,B 0,C 180,E1 -13573.322,E2 -13573.322} C_VEL
LIN {X 0,Y 360.815,Z 270.657,A -85,B 0,C 180,E1 -13573.855,E2 -13573.855} C_VEL
LIN {X 0,Y 363.682,Z 273.225,A -85,B 0,C 180,E1 -13574.591,E2 -13574.591} C_VEL
LIN {X 0,Y 366.021,Z 276.438,A -85,B 0,C 180,E1 -13575.261,E2 -13575.261} C_VEL
LIN {X 0,Y 369.29,Z 279.166,A -85,B 0,C 180,E1 -13576.185,E2 -13576.185} C_VEL
LIN {X 0,Y 372.004,Z 282.59,A -85,B 0,C 180,E1 -13577.064,E2 -13577.064} C_VEL
LIN {X 0,Y 375.164,Z 284.976,A -85,B 0,C 180,E1 -13578.108,E2 -13578.108} C_VEL
LIN {X 0,Y 378.46,Z 288.827,A -85,B 0,C 180,E1 -13579.366,E2 -13579.366} C_VEL
LIN {X 0,Y 381.679,Z 291.189,A -85,B 0,C 180,E1 -13580.702,E2 -13580.702} C_VEL
LIN {X 0,Y 383.275,Z 292.165,A -85,B 0,C 180,E1 -13581.432,E2 -13581.432} C_VEL
LIN {X 0,Y 385.674,Z 295.128,A -85,B 0,C 180,E1 -13582.76,E2 -13582.76} C_VEL
LIN {X 0,Y 387.806,Z 297.089,A -85,B 0,C 180,E1 -13584.166,E2 -13584.166} C_VEL
LIN {X 0,Y 389.864,Z 298.235,A -85,B 0,C 180,E1 -13585.865,E2 -13585.865} C_VEL
LIN {X 0,Y 391.49,Z 298.634,A -85,B 0,C 180,E1 -13587.942,E2 -13587.942} C_VEL
LIN {X 0,Y 391.908,Z 298.672,A -85,B 0,C 180,E1 -13588.972,E2 -13588.972} C_VEL
LIN {X 0,Y 392.046,Z 298.693,A -85,B 0,C 180,E1 -13590,E2 -13590} C_VEL
LIN {X 0,Y 391.908,Z 298.676,A -85,B 0,C 180,E1 -13591.028,E2 -13591.028} C_VEL
LIN {X 0,Y 391.49,Z 298.626,A -85,B 0,C 180,E1 -13592.058,E2 -13592.058} C_VEL
LIN {X 0,Y 389.864,Z 298.237,A -85,B 0,C 180,E1 -13594.135,E2 -13594.135} C_VEL
LIN {X 0,Y 387.806,Z 297.09,A -85,B 0,C 180,E1 -13595.833,E2 -13595.833} C_VEL
LIN {X 0,Y 385.677,Z 295.145,A -85,B 0,C 180,E1 -13597.238,E2 -13597.238} C_VEL
LIN {X 0,Y 383.175,Z 292.022,A -85,B 0,C 180,E1 -13598.62,E2 -13598.62} C_VEL
LIN {X 0,Y 379.709,Z 289.904,A -85,B 0,C 180,E1 -13600.127,E2 -13600.127} C_VEL
LIN {X 0,Y 376.741,Z 286.926,A -85,B 0,C 180,E1 -13601.311,E2 -13601.311} C_VEL
LIN {X 0,Y 375.158,Z 285.019,A -85,B 0,C 180,E1 -13601.892,E2 -13601.892} C_VEL
LIN {X 0,Y 371.868,Z 282.456,A -85,B 0,C 180,E1 -13602.978,E2 -13602.978} C_VEL
LIN {X 0,Y 368.721,Z 278.579,A -85,B 0,C 180,E1 -13603.984,E2 -13603.984} C_VEL
LIN {X 0,Y 365.67,Z 276.032,A -85,B 0,C 180,E1 -13604.84,E2 -13604.84} C_VEL
LIN {X 0,Y 363.068,Z 272.627,A -85,B 0,C 180,E1 -13605.568,E2 -13605.568} C_VEL
LIN {X 0,Y 360.338,Z 270.085,A -85,B 0,C 180,E1 -13606.272,E2 -13606.272} C_VEL
LIN {X 0,Y 358.398,Z 267.101,A -85,B 0,C 180,E1 -13606.783,E2 -13606.783} C_VEL
LIN {X 0,Y 356.236,Z 265.222,A -85,B 0,C 180,E1 -13607.286,E2 -13607.286} C_VEL
LIN {X 0,Y 355.046,Z 262.751,A -85,B 0,C 180,E1 -13607.609,E2 -13607.609} C_VEL
LIN {X 0,Y 354.867,Z 261.783,A -85,B 0,C 180,E1 -13607.696,E2 -13607.696} C_VEL
LIN {X 0,Y 354.831,Z 261.783,A -85,B 0,C 180,E1 -13611.45,E2 -13611.45} C_VEL
LIN {X 0,Y 354.82,Z 261.787,A -85,B 0,C 180,E1 -13614.579,E2 -13614.579} C_VEL
LIN {X 0,Y 354.829,Z 261.783,A -85,B 0,C 180,E1 -13617.1,E2 -13617.1} C_VEL
LIN {X 0,Y 354.801,Z 261.788,A -85,B 0,C 180,E1 -13619.683,E2 -13619.683} C_VEL
LIN {X 0,Y 354.78,Z 261.792,A -85,B 0,C 180,E1 -13623.687,E2 -13623.687} C_VEL
LIN {X 0,Y 354.749,Z 261.794,A -85,B 0,C 180,E1 -13626.465,E2 -13626.465} C_VEL
LIN {X 0,Y 354.777,Z 261.791,A -85,B 0,C 180,E1 -13629.429,E2 -13629.429} C_VEL
LIN {X 0,Y 354.797,Z 261.787,A -85,B 0,C 180,E1 -13632.882,E2 -13632.882} C_VEL
LIN {X 0,Y 354.823,Z 261.785,A -85,B 0,C 180,E1 -13636.125,E2 -13636.125} C_VEL
LIN {X 0,Y 354.788,Z 261.787,A -85,B 0,C 180,E1 -13639.556,E2 -13639.556} C_VEL
LIN {X 0,Y 354.76,Z 261.796,A -85,B 0,C 180,E1 -13643.547,E2 -13643.547} C_VEL
LIN {X 0,Y 354.778,Z 261.789,A -85,B 0,C 180,E1 -13644.491,E2 -13644.491} C_VEL
LIN {X 0,Y 354.087,Z 261.88,A -85,B 0,C 180,E1 -13645.439,E2 -13645.439} C_VEL
LIN {X 0,Y 351.194,Z 262.238,A -85,B 0,C 180,E1 -13646.978,E2 -13646.978} C_VEL
LIN {X 0,Y 348.775,Z 262.537,A -85,B 0,C 180,E1 -13648.224,E2 -13648.224} C_VEL
LIN {X 0,Y 347.772,Z 262.667,A -85,B 0,C 180,E1 -13649.189,E2 -13649.189} C_VEL
LIN {X 0,Y 347.708,Z 262.67,A -85,B 0,C 180,E1 -13649.516,E2 -13649.516} C_VEL
LIN {X 0,Y 347.821,Z 262.658,A -85,B 0,C 180,E1 -13652.752,E2 -13652.752} C_VEL
LIN {X 0,Y 347.76,Z 262.663,A -85,B 0,C 180,E1 -13656.169,E2 -13656.169} C_VEL
LIN {X 0,Y 347.781,Z 262.66,A -85,B 0,C 180,E1 -13659.916,E2 -13659.916} C_VEL
LIN {X 0,Y 347.812,Z 262.657,A -85,B 0,C 180,E1 -13663.575,E2 -13663.575} C_VEL
LIN {X 0,Y 347.873,Z 262.651,A -85,B 0,C 180,E1 -13667.168,E2 -13667.168} C_VEL
LIN {X 0,Y 347.922,Z 262.648,A -85,B 0,C 180,E1 -13670.708,E2 -13670.708} C_VEL
LIN {X 0,Y 348.061,Z 262.627,A -85,B 0,C 180,E1 -13673.049,E2 -13673.049} C_VEL
LIN {X 0,Y 348.187,Z 262.609,A -85,B 0,C 180,E1 -13677.693,E2 -13677.693} C_VEL
LIN {X 0,Y 348.134,Z 262.617,A -85,B 0,C 180,E1 -13681.163,E2 -13681.163} C_VEL
LIN {X 0,Y 348.181,Z 262.616,A -85,B 0,C 180,E1 -13682.32,E2 -13682.32} C_VEL
LIN {X 0,Y 348.049,Z 262.627,A -85,B 0,C 180,E1 -13686.965,E2 -13686.965} C_VEL
LIN {X 0,Y 347.895,Z 262.648,A -85,B 0,C 180,E1 -13690.482,E2 -13690.482} C_VEL
LIN {X 0,Y 347.882,Z 262.652,A -85,B 0,C 180,E1 -13694.143,E2 -13694.143} C_VEL
LIN {X 0,Y 347.799,Z 262.66,A -85,B 0,C 180,E1 -13698.247,E2 -13698.247} C_VEL
LIN {X 0,Y 347.769,Z 262.668,A -85,B 0,C 180,E1 -13701.629,E2 -13701.629} C_VEL
LIN {X 0,Y 347.741,Z 262.668,A -85,B 0,C 180,E1 -13705.12,E2 -13705.12} C_VEL
LIN {X 0,Y 347.733,Z 262.671,A -85,B 0,C 180,E1 -13707.706,E2 -13707.706} C_VEL
LIN {X 0,Y 347.745,Z 262.666,A -85,B 0,C 180,E1 -13710.354,E2 -13710.354} C_VEL
LIN {X 0,Y 347.759,Z 262.667,A -85,B 0,C 180,E1 -13714.048,E2 -13714.048} C_VEL
LIN {X 0,Y 347.777,Z 262.665,A -85,B 0,C 180,E1 -13716.068,E2 -13716.068} C_VEL
LIN {X 0,Y 348.162,Z 265.524,A -85,B 0,C 180,E1 -13719.91,E2 -13719.91} C_VEL
LIN {X 0,Y 348.624,Z 268.494,A -85,B 0,C 180,E1 -13723.471,E2 -13723.471} C_VEL
LIN {X 0,Y 348.92,Z 271.544,A -85,B 0,C 180,E1 -13726.779,E2 -13726.779} C_VEL
LIN {X 0,Y 348.854,Z 274.646,A -85,B 0,C 180,E1 -13729.86,E2 -13729.86} C_VEL
LIN {X 0,Y 348.456,Z 277.802,A -85,B 0,C 180,E1 -13732.767,E2 -13732.767} C_VEL
LIN {X 0,Y 348.042,Z 281.359,A -85,B 0,C 180,E1 -13735.892,E2 -13735.892} C_VEL
LIN {X 0,Y 347.731,Z 284.221,A -85,B 0,C 180,E1 -13738.3,E2 -13738.3} C_VEL
LIN {X 0,Y 347.232,Z 289.131,A -85,B 0,C 180,E1 -13742.257,E2 -13742.257} C_VEL
LIN {X 0,Y 346.828,Z 294.072,A -85,B 0,C 180,E1 -13746.092,E2 -13746.092} C_VEL
LIN {X 0,Y 346.598,Z 298.036,A -85,B 0,C 180,E1 -13749.088,E2 -13749.088} C_VEL
LIN {X 0,Y 348.813,Z 308.148,A -85,B 0,C 180,E1 -13749.594,E2 -13749.594} C_VEL
LIN {X 0,Y 350.611,Z 317.534,A -85,B 0,C 180,E1 -13750.177,E2 -13750.177} C_VEL
LIN {X 0,Y 351.956,Z 326.681,A -85,B 0,C 180,E1 -13750.848,E2 -13750.848} C_VEL
LIN {X 0,Y 352.948,Z 335.118,A -85,B 0,C 180,E1 -13751.573,E2 -13751.573} C_VEL
LIN {X 0,Y 352.128,Z 344.4,A -85,B 0,C 180,E1 -13752.43,E2 -13752.43} C_VEL
LIN {X 0,Y 351.135,Z 353.347,A -85,B 0,C 180,E1 -13753.429,E2 -13753.429} C_VEL
LIN {X 0,Y 350.22,Z 362.022,A -85,B 0,C 180,E1 -13754.602,E2 -13754.602} C_VEL
LIN {X 0,Y 349.426,Z 369.105,A -85,B 0,C 180,E1 -13755.737,E2 -13755.737} C_VEL
LIN {X 0,Y 348.654,Z 375.309,A -85,B 0,C 180,E1 -13756.893,E2 -13756.893} C_VEL
LIN {X 0,Y 347.806,Z 381.847,A -85,B 0,C 180,E1 -13758.342,E2 -13758.342} C_VEL
LIN {X 0,Y 347.356,Z 386.353,A -85,B 0,C 180,E1 -13759.508,E2 -13759.508} C_VEL
LIN {X 0,Y 346.776,Z 391.847,A -85,B 0,C 180,E1 -13761.257,E2 -13761.257} C_VEL
LIN {X 0,Y 346.401,Z 396.175,A -85,B 0,C 180,E1 -13763.008,E2 -13763.008} C_VEL
LIN {X 0,Y 346.268,Z 398.544,A -85,B 0,C 180,E1 -13764.176,E2 -13764.176} C_VEL
LIN {X 0,Y 346.201,Z 400.345,A -85,B 0,C 180,E1 -13765.342,E2 -13765.342} C_VEL
LIN {X 0,Y 346.091,Z 402.791,A -85,B 0,C 180,E1 -13767.672,E2 -13767.672} C_VEL
LIN {X 0,Y 346.102,Z 403.381,A -85,B 0,C 180,E1 -13768.836,E2 -13768.836} C_VEL
LIN {X 0,Y 346.102,Z 403.381,A -85,B 0,C 180,E1 -13771.164,E2 -13771.164} C_VEL
LIN {X 0,Y 346.091,Z 402.791,A -85,B 0,C 180,E1 -13772.328,E2 -13772.328} C_VEL
LIN {X 0,Y 346.201,Z 400.345,A -85,B 0,C 180,E1 -13774.658,E2 -13774.658} C_VEL
LIN {X 0,Y 346.311,Z 397.393,A -85,B 0,C 180,E1 -13776.408,E2 -13776.408} C_VEL
LIN {X 0,Y 346.631,Z 393.402,A -85,B 0,C 180,E1 -13778.159,E2 -13778.159} C_VEL
LIN {X 0,Y 347.123,Z 388.269,A -85,B 0,C 180,E1 -13779.909,E2 -13779.909} C_VEL
LIN {X 0,Y 347.692,Z 383.004,A -85,B 0,C 180,E1 -13781.366,E2 -13781.366} C_VEL
LIN {X 0,Y 348.473,Z 376.685,A -85,B 0,C 180,E1 -13782.817,E2 -13782.817} C_VEL
LIN {X 0,Y 349.195,Z 370.732,A -85,B 0,C 180,E1 -13783.976,E2 -13783.976} C_VEL
LIN {X 0,Y 350.023,Z 363.802,A -85,B 0,C 180,E1 -13785.13,E2 -13785.13} C_VEL
LIN {X 0,Y 350.858,Z 355.616,A -85,B 0,C 180,E1 -13786.286,E2 -13786.286} C_VEL
LIN {X 0,Y 351.83,Z 347.104,A -85,B 0,C 180,E1 -13787.285,E2 -13787.285} C_VEL
LIN {X 0,Y 352.769,Z 338.387,A -85,B 0,C 180,E1 -13788.136,E2 -13788.136} C_VEL
LIN {X 0,Y 352.791,Z 333.474,A -85,B 0,C 180,E1 -13788.586,E2 -13788.586} C_VEL
LIN {X 0,Y 351.316,Z 321.73,A -85,B 0,C 180,E1 -13789.536,E2 -13789.536} C_VEL
LIN {X 0,Y 349.227,Z 310.03,A -85,B 0,C 180,E1 -13790.299,E2 -13790.299} C_VEL
LIN {X 0,Y 346.779,Z 299.348,A -85,B 0,C 180,E1 -13790.863,E2 -13790.863} C_VEL
LIN {X 0,Y 346.602,Z 297.96,A -85,B 0,C 180,E1 -13790.939,E2 -13790.939} C_VEL
LIN {X 0,Y 346.924,Z 292.413,A -85,B 0,C 180,E1 -13795.177,E2 -13795.177} C_VEL
LIN {X 0,Y 347.233,Z 289.131,A -85,B 0,C 180,E1 -13797.743,E2 -13797.743} C_VEL
LIN {X 0,Y 347.732,Z 284.221,A -85,B 0,C 180,E1 -13801.7,E2 -13801.7} C_VEL
LIN {X 0,Y 348.084,Z 280.99,A -85,B 0,C 180,E1 -13804.425,E2 -13804.425} C_VEL
LIN {X 0,Y 348.621,Z 276.765,A -85,B 0,C 180,E1 -13808.16,E2 -13808.16} C_VEL
LIN {X 0,Y 348.852,Z 274.645,A -85,B 0,C 180,E1 -13810.14,E2 -13810.14} C_VEL
LIN {X 0,Y 348.966,Z 271.538,A -85,B 0,C 180,E1 -13813.214,E2 -13813.214} C_VEL
LIN {X 0,Y 348.622,Z 268.478,A -85,B 0,C 180,E1 -13816.529,E2 -13816.529} C_VEL
LIN {X 0,Y 348.165,Z 265.519,A -85,B 0,C 180,E1 -13820.089,E2 -13820.089} C_VEL
LIN {X 0,Y 347.777,Z 262.667,A -85,B 0,C 180,E1 -13823.932,E2 -13823.932} C_VEL
LIN {X 0,Y 347.735,Z 262.671,A -85,B 0,C 180,E1 -13826.922,E2 -13826.922} C_VEL
LIN {X 0,Y 347.758,Z 262.668,A -85,B 0,C 180,E1 -13830.342,E2 -13830.342} C_VEL
LIN {X 0,Y 347.74,Z 262.666,A -85,B 0,C 180,E1 -13833.594,E2 -13833.594} C_VEL
LIN {X 0,Y 347.755,Z 262.668,A -85,B 0,C 180,E1 -13836.154,E2 -13836.154} C_VEL
LIN {X 0,Y 347.776,Z 262.664,A -85,B 0,C 180,E1 -13839.901,E2 -13839.901} C_VEL
LIN {X 0,Y 347.8,Z 262.659,A -85,B 0,C 180,E1 -13843.561,E2 -13843.561} C_VEL
LIN {X 0,Y 347.888,Z 262.647,A -85,B 0,C 180,E1 -13847.154,E2 -13847.154} C_VEL
LIN {X 0,Y 347.934,Z 262.642,A -85,B 0,C 180,E1 -13850.694,E2 -13850.694} C_VEL
LIN {X 0,Y 348.032,Z 262.632,A -85,B 0,C 180,E1 -13854.199,E2 -13854.199} C_VEL
LIN {X 0,Y 348.181,Z 262.616,A -85,B 0,C 180,E1 -13857.68,E2 -13857.68} C_VEL
LIN {X 0,Y 348.109,Z 262.62,A -85,B 0,C 180,E1 -13861.15,E2 -13861.15} C_VEL
LIN {X 0,Y 348.187,Z 262.609,A -85,B 0,C 180,E1 -13862.307,E2 -13862.307} C_VEL
LIN {X 0,Y 348.061,Z 262.627,A -85,B 0,C 180,E1 -13866.951,E2 -13866.951} C_VEL
LIN {X 0,Y 347.881,Z 262.648,A -85,B 0,C 180,E1 -13870.468,E2 -13870.468} C_VEL
LIN {X 0,Y 347.882,Z 262.648,A -85,B 0,C 180,E1 -13874.143,E2 -13874.143} C_VEL
LIN {X 0,Y 347.808,Z 262.657,A -85,B 0,C 180,E1 -13878.252,E2 -13878.252} C_VEL
LIN {X 0,Y 347.744,Z 262.666,A -85,B 0,C 180,E1 -13881.619,E2 -13881.619} C_VEL
LIN {X 0,Y 347.785,Z 262.664,A -85,B 0,C 180,E1 -13885.101,E2 -13885.101} C_VEL
LIN {X 0,Y 347.779,Z 262.661,A -85,B 0,C 180,E1 -13887.687,E2 -13887.687} C_VEL
LIN {X 0,Y 347.718,Z 262.671,A -85,B 0,C 180,E1 -13890.341,E2 -13890.341} C_VEL
LIN {X 0,Y 347.714,Z 262.67,A -85,B 0,C 180,E1 -13894.037,E2 -13894.037} C_VEL
LIN {X 0,Y 347.723,Z 262.668,A -85,B 0,C 180,E1 -13897.314,E2 -13897.314} C_VEL
LIN {X 0,Y 347.754,Z 262.668,A -85,B 0,C 180,E1 -13900.282,E2 -13900.282} C_VEL
LIN {X 0,Y 347.777,Z 262.661,A -85,B 0,C 180,E1 -13903.387,E2 -13903.387} C_VEL
LIN {X 0,Y 347.773,Z 262.664,A -85,B 0,C 180,E1 -13906.664,E2 -13906.664} C_VEL
LIN {X 0,Y 347.739,Z 262.672,A -85,B 0,C 180,E1 -13910.16,E2 -13910.16} C_VEL
LIN {X 0,Y 347.738,Z 262.672,A -85,B 0,C 180,E1 -13914.12,E2 -13914.12} C_VEL
LIN {X 0,Y 347.711,Z 262.672,A -85,B 0,C 180,E1 -13918.298,E2 -13918.298} C_VEL
LIN {X 0,Y 347.752,Z 262.665,A -85,B 0,C 180,E1 -13920.986,E2 -13920.986} C_VEL
LIN {X 0,Y 347.777,Z 262.666,A -85,B 0,C 180,E1 -13923.604,E2 -13923.604} C_VEL
LIN {X 0,Y 347.782,Z 262.664,A -85,B 0,C 180,E1 -13927.422,E2 -13927.422} C_VEL
LIN {X 0,Y 347.794,Z 262.684,A -85,B 0,C 180,E1 -13931.022,E2 -13931.022} C_VEL
LIN {X 0,Y 348.589,Z 265.167,A -85,B 0,C 180,E1 -13931.242,E2 -13931.242} C_VEL
LIN {X 0,Y 350.497,Z 267.39,A -85,B 0,C 180,E1 -13931.663,E2 -13931.663} C_VEL
LIN {X 0,Y 351.478,Z 268.267,A -85,B 0,C 180,E1 -13931.874,E2 -13931.874} C_VEL
LIN {X 0,Y 353.528,Z 271.426,A -85,B 0,C 180,E1 -13932.358,E2 -13932.358} C_VEL
LIN {X 0,Y 356.02,Z 273.942,A -85,B 0,C 180,E1 -13932.947,E2 -13932.947} C_VEL
LIN {X 0,Y 358.675,Z 277.317,A -85,B 0,C 180,E1 -13933.601,E2 -13933.601} C_VEL
LIN {X 0,Y 361.179,Z 279.719,A -85,B 0,C 180,E1 -13934.245,E2 -13934.245} C_VEL
LIN {X 0,Y 364.312,Z 283.364,A -85,B 0,C 180,E1 -13935.085,E2 -13935.085} C_VEL
LIN {X 0,Y 367.066,Z 285.667,A -85,B 0,C 180,E1 -13935.849,E2 -13935.849} C_VEL
LIN {X 0,Y 370.221,Z 289.329,A -85,B 0,C 180,E1 -13936.833,E2 -13936.833} C_VEL
LIN {X 0,Y 373.849,Z 292.167,A -85,B 0,C 180,E1 -13938,E2 -13938} C_VEL
LIN {X 0,Y 376.831,Z 295.538,A -85,B 0,C 180,E1 -13939.115,E2 -13939.115} C_VEL
LIN {X 0,Y 380.396,Z 298.104,A -85,B 0,C 180,E1 -13940.551,E2 -13940.551} C_VEL
LIN {X 0,Y 381.933,Z 299.085,A -85,B 0,C 180,E1 -13941.235,E2 -13941.235} C_VEL
LIN {X 0,Y 384.562,Z 302.155,A -85,B 0,C 180,E1 -13942.65,E2 -13942.65} C_VEL
LIN {X 0,Y 386.894,Z 304.148,A -85,B 0,C 180,E1 -13944.153,E2 -13944.153} C_VEL
LIN {X 0,Y 388.977,Z 305.255,A -85,B 0,C 180,E1 -13945.856,E2 -13945.856} C_VEL
LIN {X 0,Y 389.935,Z 305.498,A -85,B 0,C 180,E1 -13946.901,E2 -13946.901} C_VEL
LIN {X 0,Y 390.619,Z 305.679,A -85,B 0,C 180,E1 -13947.938,E2 -13947.938} C_VEL
LIN {X 0,Y 391.042,Z 305.703,A -85,B 0,C 180,E1 -13948.97,E2 -13948.97} C_VEL
LIN {X 0,Y 391.183,Z 305.728,A -85,B 0,C 180,E1 -13950,E2 -13950} C_VEL
LIN {X 0,Y 391.042,Z 305.707,A -85,B 0,C 180,E1 -13951.03,E2 -13951.03} C_VEL
LIN {X 0,Y 390.618,Z 305.672,A -85,B 0,C 180,E1 -13952.062,E2 -13952.062} C_VEL
LIN {X 0,Y 389.479,Z 305.419,A -85,B 0,C 180,E1 -13953.656,E2 -13953.656} C_VEL
LIN {X 0,Y 387.603,Z 304.591,A -85,B 0,C 180,E1 -13955.332,E2 -13955.332} C_VEL
LIN {X 0,Y 385.17,Z 302.795,A -85,B 0,C 180,E1 -13956.975,E2 -13956.975} C_VEL
LIN {X 0,Y 382.399,Z 299.715,A -85,B 0,C 180,E1 -13958.521,E2 -13958.521} C_VEL
LIN {X 0,Y 381.449,Z 298.605,A -85,B 0,C 180,E1 -13959.001,E2 -13959.001} C_VEL
LIN {X 0,Y 378.193,Z 296.673,A -85,B 0,C 180,E1 -13960.355,E2 -13960.355} C_VEL
LIN {X 0,Y 374.812,Z 293.405,A -85,B 0,C 180,E1 -13961.642,E2 -13961.642} C_VEL
LIN {X 0,Y 373.018,Z 291.448,A -85,B 0,C 180,E1 -13962.283,E2 -13962.283} C_VEL
LIN {X 0,Y 369.463,Z 288.583,A -85,B 0,C 180,E1 -13963.406,E2 -13963.406} C_VEL
LIN {X 0,Y 366.374,Z 284.986,A -85,B 0,C 180,E1 -13964.348,E2 -13964.348} C_VEL
LIN {X 0,Y 363.05,Z 282.092,A -85,B 0,C 180,E1 -13965.251,E2 -13965.251} C_VEL
LIN {X 0,Y 360.218,Z 278.658,A -85,B 0,C 180,E1 -13966.01,E2 -13966.01} C_VEL
LIN {X 0,Y 357.161,Z 275.655,A -85,B 0,C 180,E1 -13966.762,E2 -13966.762} C_VEL
LIN {X 0,Y 355.351,Z 273.126,A -85,B 0,C 180,E1 -13967.217,E2 -13967.217} C_VEL
LIN {X 0,Y 352.695,Z 270.405,A -85,B 0,C 180,E1 -13967.83,E2 -13967.83} C_VEL
LIN {X 0,Y 351.064,Z 267.783,A -85,B 0,C 180,E1 -13968.22,E2 -13968.22} C_VEL
LIN {X 0,Y 348.88,Z 265.65,A -85,B 0,C 180,E1 -13968.689,E2 -13968.689} C_VEL
LIN {X 0,Y 347.929,Z 263.407,A -85,B 0,C 180,E1 -13968.932,E2 -13968.932} C_VEL
LIN {X 0,Y 347.783,Z 262.665,A -85,B 0,C 180,E1 -13969.017,E2 -13969.017} C_VEL
LIN {X 0,Y 347.782,Z 262.664,A -85,B 0,C 180,E1 -13972.578,E2 -13972.578} C_VEL
LIN {X 0,Y 347.777,Z 262.666,A -85,B 0,C 180,E1 -13976.396,E2 -13976.396} C_VEL
LIN {X 0,Y 347.717,Z 262.672,A -85,B 0,C 180,E1 -13980.35,E2 -13980.35} C_VEL
LIN {X 0,Y 347.697,Z 262.677,A -85,B 0,C 180,E1 -13984.049,E2 -13984.049} C_VEL
LIN {X 0,Y 347.714,Z 262.67,A -85,B 0,C 180,E1 -13987.326,E2 -13987.326} C_VEL
LIN {X 0,Y 347.747,Z 262.667,A -85,B 0,C 180,E1 -13990.294,E2 -13990.294} C_VEL
LIN {X 0,Y 347.775,Z 262.664,A -85,B 0,C 180,E1 -13993.399,E2 -13993.399} C_VEL
LIN {X 0,Y 347.775,Z 262.661,A -85,B 0,C 180,E1 -13996.676,E2 -13996.676} C_VEL
LIN {X 0,Y 347.747,Z 262.666,A -85,B 0,C 180,E1 -14000.172,E2 -14000.172} C_VEL
LIN {X 0,Y 347.752,Z 262.665,A -85,B 0,C 180,E1 -14004.131,E2 -14004.131} C_VEL
LIN {X 0,Y 347.705,Z 262.67,A -85,B 0,C 180,E1 -14008.093,E2 -14008.093} C_VEL
LIN {X 0,Y 347.708,Z 262.67,A -85,B 0,C 180,E1 -14009.516,E2 -14009.516} C_VEL
LIN {X 0,Y 347.095,Z 262.752,A -85,B 0,C 180,E1 -14010.484,E2 -14010.484} C_VEL
LIN {X 0,Y 344.281,Z 263.101,A -85,B 0,C 180,E1 -14012.059,E2 -14012.059} C_VEL
LIN {X 0,Y 341.865,Z 263.401,A -85,B 0,C 180,E1 -14013.334,E2 -14013.334} C_VEL
LIN {X 0,Y 340.821,Z 263.528,A -85,B 0,C 180,E1 -14014.32,E2 -14014.32} C_VEL
LIN {X 0,Y 340.734,Z 263.539,A -85,B 0,C 180,E1 -14014.654,E2 -14014.654} C_VEL
LIN {X 0,Y 340.718,Z 263.541,A -85,B 0,C 180,E1 -14018.214,E2 -14018.214} C_VEL
LIN {X 0,Y 340.772,Z 263.534,A -85,B 0,C 180,E1 -14021.988,E2 -14021.988} C_VEL
LIN {X 0,Y 340.835,Z 263.525,A -85,B 0,C 180,E1 -14025.724,E2 -14025.724} C_VEL
LIN {X 0,Y 340.833,Z 263.526,A -85,B 0,C 180,E1 -14029.313,E2 -14029.313} C_VEL
LIN {X 0,Y 341.03,Z 263.504,A -85,B 0,C 180,E1 -14032.905,E2 -14032.905} C_VEL
LIN {X 0,Y 341.124,Z 263.488,A -85,B 0,C 180,E1 -14037.645,E2 -14037.645} C_VEL
LIN {X 0,Y 341.102,Z 263.492,A -85,B 0,C 180,E1 -14041.187,E2 -14041.187} C_VEL
LIN {X 0,Y 341.118,Z 263.495,A -85,B 0,C 180,E1 -14042.368,E2 -14042.368} C_VEL
LIN {X 0,Y 341.008,Z 263.508,A -85,B 0,C 180,E1 -14045.921,E2 -14045.921} C_VEL
LIN {X 0,Y 340.963,Z 263.513,A -85,B 0,C 180,E1 -14048.363,E2 -14048.363} C_VEL
LIN {X 0,Y 340.849,Z 263.53,A -85,B 0,C 180,E1 -14051.906,E2 -14051.906} C_VEL
LIN {X 0,Y 340.795,Z 263.534,A -85,B 0,C 180,E1 -14055.557,E2 -14055.557} C_VEL
LIN {X 0,Y 340.708,Z 263.544,A -85,B 0,C 180,E1 -14059.277,E2 -14059.277} C_VEL
LIN {X 0,Y 340.707,Z 263.544,A -85,B 0,C 180,E1 -14063.08,E2 -14063.08} C_VEL
LIN {X 0,Y 340.717,Z 263.542,A -85,B 0,C 180,E1 -14066.993,E2 -14066.993} C_VEL
LIN {X 0,Y 340.702,Z 263.546,A -85,B 0,C 180,E1 -14071.05,E2 -14071.05} C_VEL
LIN {X 0,Y 340.726,Z 263.545,A -85,B 0,C 180,E1 -14075.284,E2 -14075.284} C_VEL
LIN {X 0,Y 340.817,Z 264.249,A -85,B 0,C 180,E1 -14076.733,E2 -14076.733} C_VEL
LIN {X 0,Y 341.194,Z 266.968,A -85,B 0,C 180,E1 -14080.348,E2 -14080.348} C_VEL
LIN {X 0,Y 341.629,Z 269.976,A -85,B 0,C 180,E1 -14083.945,E2 -14083.945} C_VEL
LIN {X 0,Y 341.9,Z 273.033,A -85,B 0,C 180,E1 -14087.287,E2 -14087.287} C_VEL
LIN {X 0,Y 341.742,Z 276.141,A -85,B 0,C 180,E1 -14090.394,E2 -14090.394} C_VEL
LIN {X 0,Y 341.299,Z 279.399,A -85,B 0,C 180,E1 -14093.432,E2 -14093.432} C_VEL
LIN {X 0,Y 340.918,Z 282.487,A -85,B 0,C 180,E1 -14096.18,E2 -14096.18} C_VEL
LIN {X 0,Y 340.404,Z 287.146,A -85,B 0,C 180,E1 -14100.135,E2 -14100.135} C_VEL
LIN {X 0,Y 340.079,Z 290.622,A -85,B 0,C 180,E1 -14102.958,E2 -14102.958} C_VEL
LIN {X 0,Y 339.814,Z 293.903,A -85,B 0,C 180,E1 -14105.567,E2 -14105.567} C_VEL
LIN {X 0,Y 339.534,Z 297.78,A -85,B 0,C 180,E1 -14108.615,E2 -14108.615} C_VEL
LIN {X 0,Y 342.663,Z 311.892,A -85,B 0,C 180,E1 -14109.387,E2 -14109.387} C_VEL
LIN {X 0,Y 344.744,Z 324.759,A -85,B 0,C 180,E1 -14110.302,E2 -14110.302} C_VEL
LIN {X 0,Y 345.965,Z 334.899,A -85,B 0,C 180,E1 -14111.187,E2 -14111.187} C_VEL
LIN {X 0,Y 345.881,Z 339.809,A -85,B 0,C 180,E1 -14111.643,E2 -14111.643} C_VEL
LIN {X 0,Y 344.445,Z 351.999,A -85,B 0,C 180,E1 -14112.944,E2 -14112.944} C_VEL
LIN {X 0,Y 343.45,Z 360.709,A -85,B 0,C 180,E1 -14114.116,E2 -14114.116} C_VEL
LIN {X 0,Y 342.501,Z 368.892,A -85,B 0,C 180,E1 -14115.442,E2 -14115.442} C_VEL
LIN {X 0,Y 341.711,Z 375.097,A -85,B 0,C 180,E1 -14116.622,E2 -14116.622} C_VEL
LIN {X 0,Y 340.826,Z 381.635,A -85,B 0,C 180,E1 -14118.1,E2 -14118.1} C_VEL
LIN {X 0,Y 340.363,Z 386.141,A -85,B 0,C 180,E1 -14119.29,E2 -14119.29} C_VEL
LIN {X 0,Y 339.74,Z 391.635,A -85,B 0,C 180,E1 -14121.075,E2 -14121.075} C_VEL
LIN {X 0,Y 339.346,Z 395.963,A -85,B 0,C 180,E1 -14122.862,E2 -14122.862} C_VEL
LIN {X 0,Y 339.189,Z 398.332,A -85,B 0,C 180,E1 -14124.054,E2 -14124.054} C_VEL
LIN {X 0,Y 339.105,Z 400.133,A -85,B 0,C 180,E1 -14125.245,E2 -14125.245} C_VEL
LIN {X 0,Y 339.006,Z 402.58,A -85,B 0,C 180,E1 -14127.624,E2 -14127.624} C_VEL
LIN {X 0,Y 339.006,Z 403.17,A -85,B 0,C 180,E1 -14128.812,E2 -14128.812} C_VEL
LIN {X 0,Y 339.006,Z 403.17,A -85,B 0,C 180,E1 -14131.188,E2 -14131.188} C_VEL
LIN {X 0,Y 339.006,Z 402.58,A -85,B 0,C 180,E1 -14132.376,E2 -14132.376} C_VEL
LIN {X 0,Y 339.105,Z 400.133,A -85,B 0,C 180,E1 -14134.755,E2 -14134.755} C_VEL
LIN {X 0,Y 339.251,Z 397.181,A -85,B 0,C 180,E1 -14136.542,E2 -14136.542} C_VEL
LIN {X 0,Y 339.584,Z 393.19,A -85,B 0,C 180,E1 -14138.33,E2 -14138.33} C_VEL
LIN {X 0,Y 340.112,Z 388.057,A -85,B 0,C 180,E1 -14140.116,E2 -14140.116} C_VEL
LIN {X 0,Y 340.681,Z 382.791,A -85,B 0,C 180,E1 -14141.603,E2 -14141.603} C_VEL
LIN {X 0,Y 341.517,Z 376.473,A -85,B 0,C 180,E1 -14143.083,E2 -14143.083} C_VEL
LIN {X 0,Y 342.267,Z 370.519,A -85,B 0,C 180,E1 -14144.265,E2 -14144.265} C_VEL
LIN {X 0,Y 343.282,Z 362.491,A -85,B 0,C 180,E1 -14145.609,E2 -14145.609} C_VEL
LIN {X 0,Y 344.156,Z 354.269,A -85,B 0,C 180,E1 -14146.765,E2 -14146.765} C_VEL
LIN {X 0,Y 345.229,Z 345.541,A -85,B 0,C 180,E1 -14147.78,E2 -14147.78} C_VEL
LIN {X 0,Y 346.102,Z 336.541,A -85,B 0,C 180,E1 -14148.652,E2 -14148.652} C_VEL
LIN {X 0,Y 345.069,Z 327.217,A -85,B 0,C 180,E1 -14149.491,E2 -14149.491} C_VEL
LIN {X 0,Y 343.855,Z 318.814,A -85,B 0,C 180,E1 -14150.139,E2 -14150.139} C_VEL
LIN {X 0,Y 341.973,Z 308.732,A -85,B 0,C 180,E1 -14150.797,E2 -14150.797} C_VEL
LIN {X 0,Y 339.707,Z 299.218,A -85,B 0,C 180,E1 -14151.315,E2 -14151.315} C_VEL
LIN {X 0,Y 339.535,Z 297.78,A -85,B 0,C 180,E1 -14151.385,E2 -14151.385} C_VEL
LIN {X 0,Y 339.804,Z 293.843,A -85,B 0,C 180,E1 -14154.482,E2 -14154.482} C_VEL
LIN {X 0,Y 340.228,Z 288.995,A -85,B 0,C 180,E1 -14158.366,E2 -14158.366} C_VEL
LIN {X 0,Y 340.734,Z 284.095,A -85,B 0,C 180,E1 -14162.43,E2 -14162.43} C_VEL
LIN {X 0,Y 341.147,Z 280.878,A -85,B 0,C 180,E1 -14165.227,E2 -14165.227} C_VEL
LIN {X 0,Y 341.635,Z 277.218,A -85,B 0,C 180,E1 -14168.575,E2 -14168.575} C_VEL
LIN {X 0,Y 341.883,Z 274.575,A -85,B 0,C 180,E1 -14171.133,E2 -14171.133} C_VEL
LIN {X 0,Y 341.873,Z 271.825,A -85,B 0,C 180,E1 -14173.98,E2 -14173.98} C_VEL
LIN {X 0,Y 341.476,Z 268.966,A -85,B 0,C 180,E1 -14177.214,E2 -14177.214} C_VEL
LIN {X 0,Y 341.121,Z 266.467,A -85,B 0,C 180,E1 -14180.3,E2 -14180.3} C_VEL
LIN {X 0,Y 340.8,Z 264.055,A -85,B 0,C 180,E1 -14183.537,E2 -14183.537} C_VEL
LIN {X 0,Y 340.726,Z 263.546,A -85,B 0,C 180,E1 -14184.716,E2 -14184.716} C_VEL
LIN {X 0,Y 340.702,Z 263.546,A -85,B 0,C 180,E1 -14188.95,E2 -14188.95} C_VEL
LIN {X 0,Y 340.717,Z 263.543,A -85,B 0,C 180,E1 -14193.007,E2 -14193.007} C_VEL
LIN {X 0,Y 340.707,Z 263.544,A -85,B 0,C 180,E1 -14196.92,E2 -14196.92} C_VEL
LIN {X 0,Y 340.708,Z 263.544,A -85,B 0,C 180,E1 -14200.723,E2 -14200.723} C_VEL
LIN {X 0,Y 340.795,Z 263.534,A -85,B 0,C 180,E1 -14204.443,E2 -14204.443} C_VEL
LIN {X 0,Y 340.849,Z 263.53,A -85,B 0,C 180,E1 -14208.094,E2 -14208.094} C_VEL
LIN {X 0,Y 340.979,Z 263.512,A -85,B 0,C 180,E1 -14211.698,E2 -14211.698} C_VEL
LIN {X 0,Y 341.008,Z 263.508,A -85,B 0,C 180,E1 -14214.079,E2 -14214.079} C_VEL
LIN {X 0,Y 341.118,Z 263.495,A -85,B 0,C 180,E1 -14217.632,E2 -14217.632} C_VEL
LIN {X 0,Y 341.08,Z 263.495,A -85,B 0,C 180,E1 -14221.174,E2 -14221.174} C_VEL
LIN {X 0,Y 341.124,Z 263.488,A -85,B 0,C 180,E1 -14222.355,E2 -14222.355} C_VEL
LIN {X 0,Y 341.03,Z 263.504,A -85,B 0,C 180,E1 -14227.095,E2 -14227.095} C_VEL
LIN {X 0,Y 340.833,Z 263.526,A -85,B 0,C 180,E1 -14230.687,E2 -14230.687} C_VEL
LIN {X 0,Y 340.846,Z 263.524,A -85,B 0,C 180,E1 -14234.318,E2 -14234.318} C_VEL
LIN {X 0,Y 340.765,Z 263.535,A -85,B 0,C 180,E1 -14238.433,E2 -14238.433} C_VEL
LIN {X 0,Y 340.694,Z 263.544,A -85,B 0,C 180,E1 -14241.834,E2 -14241.834} C_VEL
LIN {X 0,Y 340.745,Z 263.537,A -85,B 0,C 180,E1 -14245.657,E2 -14245.657} C_VEL
LIN {X 0,Y 340.699,Z 263.544,A -85,B 0,C 180,E1 -14248.314,E2 -14248.314} C_VEL
LIN {X 0,Y 340.666,Z 263.55,A -85,B 0,C 180,E1 -14251.038,E2 -14251.038} C_VEL
LIN {X 0,Y 340.682,Z 263.546,A -85,B 0,C 180,E1 -14255.272,E2 -14255.272} C_VEL
LIN {X 0,Y 340.672,Z 263.551,A -85,B 0,C 180,E1 -14258.379,E2 -14258.379} C_VEL
LIN {X 0,Y 340.685,Z 263.545,A -85,B 0,C 180,E1 -14261.297,E2 -14261.297} C_VEL
LIN {X 0,Y 340.738,Z 263.542,A -85,B 0,C 180,E1 -14264.516,E2 -14264.516} C_VEL
LIN {X 0,Y 340.706,Z 263.545,A -85,B 0,C 180,E1 -14267.939,E2 -14267.939} C_VEL
LIN {X 0,Y 340.687,Z 263.55,A -85,B 0,C 180,E1 -14270.247,E2 -14270.247} C_VEL
LIN {X 0,Y 340.661,Z 263.549,A -85,B 0,C 180,E1 -14273.554,E2 -14273.554} C_VEL
LIN {X 0,Y 340.644,Z 263.555,A -85,B 0,C 180,E1 -14276.149,E2 -14276.149} C_VEL
LIN {X 0,Y 340.722,Z 263.542,A -85,B 0,C 180,E1 -14280.328,E2 -14280.328} C_VEL
LIN {X 0,Y 340.75,Z 263.537,A -85,B 0,C 180,E1 -14283.016,E2 -14283.016} C_VEL
LIN {X 0,Y 340.735,Z 263.54,A -85,B 0,C 180,E1 -14286.928,E2 -14286.928} C_VEL
LIN {X 0,Y 340.74,Z 263.543,A -85,B 0,C 180,E1 -14289.829,E2 -14289.829} C_VEL
LIN {X 0,Y 341.787,Z 266.447,A -85,B 0,C 180,E1 -14290.105,E2 -14290.105} C_VEL
LIN {X 0,Y 344.192,Z 269.124,A -85,B 0,C 180,E1 -14290.587,E2 -14290.587} C_VEL
LIN {X 0,Y 346.227,Z 272.189,A -85,B 0,C 180,E1 -14291.025,E2 -14291.025} C_VEL
LIN {X 0,Y 348.316,Z 274.351,A -85,B 0,C 180,E1 -14291.468,E2 -14291.468} C_VEL
LIN {X 0,Y 350.834,Z 277.769,A -85,B 0,C 180,E1 -14292.046,E2 -14292.046} C_VEL
LIN {X 0,Y 353.147,Z 280.076,A -85,B 0,C 180,E1 -14292.553,E2 -14292.553} C_VEL
LIN {X 0,Y 356.483,Z 283.981,A -85,B 0,C 180,E1 -14293.367,E2 -14293.367} C_VEL
LIN {X 0,Y 358.758,Z 286.159,A -85,B 0,C 180,E1 -14293.912,E2 -14293.912} C_VEL
LIN {X 0,Y 362.117,Z 289.871,A -85,B 0,C 180,E1 -14294.804,E2 -14294.804} C_VEL
LIN {X 0,Y 364.957,Z 292.307,A -85,B 0,C 180,E1 -14295.564,E2 -14295.564} C_VEL
LIN {X 0,Y 368.542,Z 296.124,A -85,B 0,C 180,E1 -14296.63,E2 -14296.63} C_VEL
LIN {X 0,Y 372.231,Z 299.122,A -85,B 0,C 180,E1 -14297.799,E2 -14297.799} C_VEL
LIN {X 0,Y 375.545,Z 302.562,A -85,B 0,C 180,E1 -14299.009,E2 -14299.009} C_VEL
LIN {X 0,Y 379.044,Z 305.001,A -85,B 0,C 180,E1 -14300.394,E2 -14300.394} C_VEL
LIN {X 0,Y 380.473,Z 305.946,A -85,B 0,C 180,E1 -14301.023,E2 -14301.023} C_VEL
LIN {X 0,Y 383.294,Z 309.171,A -85,B 0,C 180,E1 -14302.55,E2 -14302.55} C_VEL
LIN {X 0,Y 385.773,Z 311.18,A -85,B 0,C 180,E1 -14304.135,E2 -14304.135} C_VEL
LIN {X 0,Y 387.882,Z 312.269,A -85,B 0,C 180,E1 -14305.844,E2 -14305.844} C_VEL
LIN {X 0,Y 388.852,Z 312.514,A -85,B 0,C 180,E1 -14306.892,E2 -14306.892} C_VEL
LIN {X 0,Y 389.529,Z 312.694,A -85,B 0,C 180,E1 -14307.932,E2 -14307.932} C_VEL
LIN {X 0,Y 389.958,Z 312.719,A -85,B 0,C 180,E1 -14308.967,E2 -14308.967} C_VEL
LIN {X 0,Y 390.105,Z 312.745,A -85,B 0,C 180,E1 -14310,E2 -14310} C_VEL
LIN {X 0,Y 389.536,Z 312.661,A -85,B 0,C 180,E1 -14312.068,E2 -14312.068} C_VEL
LIN {X 0,Y 388.36,Z 312.43,A -85,B 0,C 180,E1 -14313.667,E2 -14313.667} C_VEL
LIN {X 0,Y 386.379,Z 311.526,A -85,B 0,C 180,E1 -14315.439,E2 -14315.439} C_VEL
LIN {X 0,Y 383.749,Z 309.601,A -85,B 0,C 180,E1 -14317.183,E2 -14317.183} C_VEL
LIN {X 0,Y 380.976,Z 306.568,A -85,B 0,C 180,E1 -14318.718,E2 -14318.718} C_VEL
LIN {X 0,Y 379.638,Z 305.29,A -85,B 0,C 180,E1 -14319.345,E2 -14319.345} C_VEL
LIN {X 0,Y 376.352,Z 303.205,A -85,B 0,C 180,E1 -14320.686,E2 -14320.686} C_VEL
LIN {X 0,Y 372.813,Z 299.802,A -85,B 0,C 180,E1 -14322.001,E2 -14322.001} C_VEL
LIN {X 0,Y 371.154,Z 298.105,A -85,B 0,C 180,E1 -14322.559,E2 -14322.559} C_VEL
LIN {X 0,Y 367.31,Z 295.006,A -85,B 0,C 180,E1 -14323.738,E2 -14323.738} C_VEL
LIN {X 0,Y 363.886,Z 291.244,A -85,B 0,C 180,E1 -14324.738,E2 -14324.738} C_VEL
LIN {X 0,Y 360.07,Z 287.837,A -85,B 0,C 180,E1 -14325.73,E2 -14325.73} C_VEL
LIN {X 0,Y 357.598,Z 284.91,A -85,B 0,C 180,E1 -14326.376,E2 -14326.376} C_VEL
LIN {X 0,Y 354.071,Z 281.391,A -85,B 0,C 180,E1 -14327.216,E2 -14327.216} C_VEL
LIN {X 0,Y 352.17,Z 278.985,A -85,B 0,C 180,E1 -14327.665,E2 -14327.665} C_VEL
LIN {X 0,Y 348.99,Z 275.487,A -85,B 0,C 180,E1 -14328.373,E2 -14328.373} C_VEL
LIN {X 0,Y 347.561,Z 273.468,A -85,B 0,C 180,E1 -14328.698,E2 -14328.698} C_VEL
LIN {X 0,Y 344.945,Z 270.526,A -85,B 0,C 180,E1 -14329.245,E2 -14329.245} C_VEL
LIN {X 0,Y 343.677,Z 268.43,A -85,B 0,C 180,E1 -14329.519,E2 -14329.519} C_VEL
LIN {X 0,Y 341.638,Z 266.195,A -85,B 0,C 180,E1 -14329.928,E2 -14329.928} C_VEL
LIN {X 0,Y 340.745,Z 263.543,A -85,B 0,C 180,E1 -14330.192,E2 -14330.192} C_VEL
LIN {X 0,Y 340.735,Z 263.54,A -85,B 0,C 180,E1 -14333.072,E2 -14333.072} C_VEL
LIN {X 0,Y 340.75,Z 263.537,A -85,B 0,C 180,E1 -14336.984,E2 -14336.984} C_VEL
LIN {X 0,Y 340.712,Z 263.546,A -85,B 0,C 180,E1 -14339.983,E2 -14339.983} C_VEL
LIN {X 0,Y 340.644,Z 263.555,A -85,B 0,C 180,E1 -14343.851,E2 -14343.851} C_VEL
LIN {X 0,Y 340.656,Z 263.549,A -85,B 0,C 180,E1 -14346.747,E2 -14346.747} C_VEL
LIN {X 0,Y 340.717,Z 263.542,A -85,B 0,C 180,E1 -14350.268,E2 -14350.268} C_VEL
LIN {X 0,Y 340.735,Z 263.543,A -85,B 0,C 180,E1 -14353.801,E2 -14353.801} C_VEL
LIN {X 0,Y 340.719,Z 263.542,A -85,B 0,C 180,E1 -14357.115,E2 -14357.115} C_VEL
LIN {X 0,Y 340.695,Z 263.544,A -85,B 0,C 180,E1 -14360.259,E2 -14360.259} C_VEL
LIN {X 0,Y 340.673,Z 263.55,A -85,B 0,C 180,E1 -14363.566,E2 -14363.566} C_VEL
LIN {X 0,Y 340.658,Z 263.548,A -85,B 0,C 180,E1 -14366.16,E2 -14366.16} C_VEL
LIN {X 0,Y 340.711,Z 263.542,A -85,B 0,C 180,E1 -14370.336,E2 -14370.336} C_VEL
LIN {X 0,Y 340.775,Z 263.539,A -85,B 0,C 180,E1 -14373.027,E2 -14373.027} C_VEL
LIN {X 0,Y 340.734,Z 263.539,A -85,B 0,C 180,E1 -14374.654,E2 -14374.654} C_VEL
LIN {X 0,Y 340.052,Z 263.627,A -85,B 0,C 180,E1 -14375.641,E2 -14375.641} C_VEL
LIN {X 0,Y 337.162,Z 263.987,A -85,B 0,C 180,E1 -14377.246,E2 -14377.246} C_VEL
LIN {X 0,Y 334.733,Z 264.288,A -85,B 0,C 180,E1 -14378.545,E2 -14378.545} C_VEL
LIN {X 0,Y 333.713,Z 264.413,A -85,B 0,C 180,E1 -14379.551,E2 -14379.551} C_VEL
LIN {X 0,Y 333.642,Z 264.421,A -85,B 0,C 180,E1 -14379.892,E2 -14379.892} C_VEL
LIN {X 0,Y 333.699,Z 264.42,A -85,B 0,C 180,E1 -14382.86,E2 -14382.86} C_VEL
LIN {X 0,Y 333.776,Z 264.41,A -85,B 0,C 180,E1 -14386.616,E2 -14386.616} C_VEL
LIN {X 0,Y 333.806,Z 264.404,A -85,B 0,C 180,E1 -14390.311,E2 -14390.311} C_VEL
LIN {X 0,Y 333.991,Z 264.38,A -85,B 0,C 180,E1 -14393.968,E2 -14393.968} C_VEL
LIN {X 0,Y 334.065,Z 264.366,A -85,B 0,C 180,E1 -14397.596,E2 -14397.596} C_VEL
LIN {X 0,Y 334.071,Z 264.368,A -85,B 0,C 180,E1 -14401.212,E2 -14401.212} C_VEL
LIN {X 0,Y 334.059,Z 264.374,A -85,B 0,C 180,E1 -14402.418,E2 -14402.418} C_VEL
LIN {X 0,Y 333.982,Z 264.385,A -85,B 0,C 180,E1 -14406.046,E2 -14406.046} C_VEL
LIN {X 0,Y 333.912,Z 264.391,A -85,B 0,C 180,E1 -14408.479,E2 -14408.479} C_VEL
LIN {X 0,Y 333.79,Z 264.408,A -85,B 0,C 180,E1 -14412.161,E2 -14412.161} C_VEL
LIN {X 0,Y 333.72,Z 264.418,A -85,B 0,C 180,E1 -14415.895,E2 -14415.895} C_VEL
LIN {X 0,Y 333.7,Z 264.415,A -85,B 0,C 180,E1 -14418.609,E2 -14418.609} C_VEL
LIN {X 0,Y 333.655,Z 264.422,A -85,B 0,C 180,E1 -14422.287,E2 -14422.287} C_VEL
LIN {X 0,Y 333.663,Z 264.421,A -85,B 0,C 180,E1 -14425.082,E2 -14425.082} C_VEL
LIN {X 0,Y 333.637,Z 264.425,A -85,B 0,C 180,E1 -14428.985,E2 -14428.985} C_VEL
LIN {X 0,Y 333.652,Z 264.423,A -85,B 0,C 180,E1 -14432.591,E2 -14432.591} C_VEL
LIN {X 0,Y 333.695,Z 264.421,A -85,B 0,C 180,E1 -14434.778,E2 -14434.778} C_VEL
LIN {X 0,Y 333.813,Z 265.491,A -85,B 0,C 180,E1 -14436.867,E2 -14436.867} C_VEL
LIN {X 0,Y 334.215,Z 268.438,A -85,B 0,C 180,E1 -14440.799,E2 -14440.799} C_VEL
LIN {X 0,Y 334.665,Z 271.435,A -85,B 0,C 180,E1 -14444.439,E2 -14444.439} C_VEL
LIN {X 0,Y 334.875,Z 274.506,A -85,B 0,C 180,E1 -14447.812,E2 -14447.812} C_VEL
LIN {X 0,Y 334.619,Z 277.683,A -85,B 0,C 180,E1 -14451.003,E2 -14451.003} C_VEL
LIN {X 0,Y 334.037,Z 282.114,A -85,B 0,C 180,E1 -14455.146,E2 -14455.146} C_VEL
LIN {X 0,Y 333.561,Z 285.582,A -85,B 0,C 180,E1 -14458.215,E2 -14458.215} C_VEL
LIN {X 0,Y 333.078,Z 290.454,A -85,B 0,C 180,E1 -14462.342,E2 -14462.342} C_VEL
LIN {X 0,Y 332.609,Z 295.378,A -85,B 0,C 180,E1 -14466.33,E2 -14466.33} C_VEL
LIN {X 0,Y 332.465,Z 297.598,A -85,B 0,C 180,E1 -14468.147,E2 -14468.147} C_VEL
LIN {X 0,Y 334.963,Z 308.407,A -85,B 0,C 180,E1 -14468.742,E2 -14468.742} C_VEL
LIN {X 0,Y 336.871,Z 318.718,A -85,B 0,C 180,E1 -14469.432,E2 -14469.432} C_VEL
LIN {X 0,Y 338.253,Z 328.015,A -85,B 0,C 180,E1 -14470.179,E2 -14470.179} C_VEL
LIN {X 0,Y 339.178,Z 336.323,A -85,B 0,C 180,E1 -14470.953,E2 -14470.953} C_VEL
LIN {X 0,Y 338.792,Z 342.626,A -85,B 0,C 180,E1 -14471.558,E2 -14471.558} C_VEL
LIN {X 0,Y 337.502,Z 352.923,A -85,B 0,C 180,E1 -14472.739,E2 -14472.739} C_VEL
LIN {X 0,Y 336.476,Z 361.362,A -85,B 0,C 180,E1 -14473.919,E2 -14473.919} C_VEL
LIN {X 0,Y 335.573,Z 368.679,A -85,B 0,C 180,E1 -14475.135,E2 -14475.135} C_VEL
LIN {X 0,Y 334.786,Z 374.885,A -85,B 0,C 180,E1 -14476.34,E2 -14476.34} C_VEL
LIN {X 0,Y 333.858,Z 381.423,A -85,B 0,C 180,E1 -14477.848,E2 -14477.848} C_VEL
LIN {X 0,Y 333.354,Z 385.929,A -85,B 0,C 180,E1 -14479.062,E2 -14479.062} C_VEL
LIN {X 0,Y 332.691,Z 391.423,A -85,B 0,C 180,E1 -14480.884,E2 -14480.884} C_VEL
LIN {X 0,Y 332.285,Z 395.751,A -85,B 0,C 180,E1 -14482.709,E2 -14482.709} C_VEL
LIN {X 0,Y 332.087,Z 398.399,A -85,B 0,C 180,E1 -14484.114,E2 -14484.114} C_VEL
LIN {X 0,Y 332.009,Z 401.311,A -85,B 0,C 180,E1 -14486.359,E2 -14486.359} C_VEL
LIN {X 0,Y 331.924,Z 402.369,A -85,B 0,C 180,E1 -14487.573,E2 -14487.573} C_VEL
LIN {X 0,Y 331.913,Z 402.958,A -85,B 0,C 180,E1 -14488.787,E2 -14488.787} C_VEL
LIN {X 0,Y 331.913,Z 402.958,A -85,B 0,C 180,E1 -14491.213,E2 -14491.213} C_VEL
LIN {X 0,Y 331.924,Z 402.369,A -85,B 0,C 180,E1 -14492.427,E2 -14492.427} C_VEL
LIN {X 0,Y 332.013,Z 399.921,A -85,B 0,C 180,E1 -14494.857,E2 -14494.857} C_VEL
LIN {X 0,Y 332.186,Z 396.969,A -85,B 0,C 180,E1 -14496.682,E2 -14496.682} C_VEL
LIN {X 0,Y 332.528,Z 392.978,A -85,B 0,C 180,E1 -14498.508,E2 -14498.508} C_VEL
LIN {X 0,Y 333.093,Z 387.845,A -85,B 0,C 180,E1 -14500.331,E2 -14500.331} C_VEL
LIN {X 0,Y 333.696,Z 382.579,A -85,B 0,C 180,E1 -14501.849,E2 -14501.849} C_VEL
LIN {X 0,Y 334.576,Z 376.261,A -85,B 0,C 180,E1 -14503.359,E2 -14503.359} C_VEL
LIN {X 0,Y 335.342,Z 370.306,A -85,B 0,C 180,E1 -14504.566,E2 -14504.566} C_VEL
LIN {X 0,Y 336.388,Z 362.376,A -85,B 0,C 180,E1 -14505.922,E2 -14505.922} C_VEL
LIN {X 0,Y 337.19,Z 355.192,A -85,B 0,C 180,E1 -14506.965,E2 -14506.965} C_VEL
LIN {X 0,Y 338.3,Z 346.681,A -85,B 0,C 180,E1 -14508,E2 -14508} C_VEL
LIN {X 0,Y 339.237,Z 337.963,A -85,B 0,C 180,E1 -14508.887,E2 -14508.887} C_VEL
LIN {X 0,Y 338.363,Z 329.048,A -85,B 0,C 180,E1 -14509.734,E2 -14509.734} C_VEL
LIN {X 0,Y 336.933,Z 318.911,A -85,B 0,C 180,E1 -14510.552,E2 -14510.552} C_VEL
LIN {X 0,Y 335.086,Z 309.013,A -85,B 0,C 180,E1 -14511.222,E2 -14511.222} C_VEL
LIN {X 0,Y 332.734,Z 299.379,A -85,B 0,C 180,E1 -14511.772,E2 -14511.772} C_VEL
LIN {X 0,Y 332.443,Z 297.562,A -85,B 0,C 180,E1 -14511.884,E2 -14511.884} C_VEL
LIN {X 0,Y 332.747,Z 293.738,A -85,B 0,C 180,E1 -14514.987,E2 -14514.987} C_VEL
LIN {X 0,Y 333.078,Z 290.454,A -85,B 0,C 180,E1 -14517.658,E2 -14517.658} C_VEL
LIN {X 0,Y 333.561,Z 285.575,A -85,B 0,C 180,E1 -14521.785,E2 -14521.785} C_VEL
LIN {X 0,Y 334.04,Z 282.105,A -85,B 0,C 180,E1 -14524.854,E2 -14524.854} C_VEL
LIN {X 0,Y 334.619,Z 277.68,A -85,B 0,C 180,E1 -14528.996,E2 -14528.996} C_VEL
LIN {X 0,Y 334.896,Z 274.504,A -85,B 0,C 180,E1 -14532.185,E2 -14532.185} C_VEL
LIN {X 0,Y 334.805,Z 272.398,A -85,B 0,C 180,E1 -14534.456,E2 -14534.456} C_VEL
LIN {X 0,Y 334.415,Z 269.605,A -85,B 0,C 180,E1 -14537.733,E2 -14537.733} C_VEL
LIN {X 0,Y 334.014,Z 266.936,A -85,B 0,C 180,E1 -14541.124,E2 -14541.124} C_VEL
LIN {X 0,Y 333.765,Z 264.974,A -85,B 0,C 180,E1 -14543.866,E2 -14543.866} C_VEL
LIN {X 0,Y 333.683,Z 264.421,A -85,B 0,C 180,E1 -14545.336,E2 -14545.336} C_VEL
LIN {X 0,Y 333.638,Z 264.427,A -85,B 0,C 180,E1 -14548.217,E2 -14548.217} C_VEL
LIN {X 0,Y 333.637,Z 264.425,A -85,B 0,C 180,E1 -14551.015,E2 -14551.015} C_VEL
LIN {X 0,Y 333.663,Z 264.422,A -85,B 0,C 180,E1 -14554.918,E2 -14554.918} C_VEL
LIN {X 0,Y 333.657,Z 264.422,A -85,B 0,C 180,E1 -14559.011,E2 -14559.011} C_VEL
LIN {X 0,Y 333.716,Z 264.414,A -85,B 0,C 180,E1 -14561.579,E2 -14561.579} C_VEL
LIN {X 0,Y 333.777,Z 264.407,A -85,B 0,C 180,E1 -14565.594,E2 -14565.594} C_VEL
LIN {X 0,Y 333.817,Z 264.4,A -85,B 0,C 180,E1 -14569.071,E2 -14569.071} C_VEL
LIN {X 0,Y 333.953,Z 264.384,A -85,B 0,C 180,E1 -14572.739,E2 -14572.739} C_VEL
LIN {X 0,Y 333.772,Z 264.407,A -85,B 0,C 180,E1 -14575.162,E2 -14575.162} C_VEL
LIN {X 0,Y 334.059,Z 264.374,A -85,B 0,C 180,E1 -14577.582,E2 -14577.582} C_VEL
LIN {X 0,Y 334.051,Z 264.37,A -85,B 0,C 180,E1 -14581.198,E2 -14581.198} C_VEL
LIN {X 0,Y 334.065,Z 264.366,A -85,B 0,C 180,E1 -14582.404,E2 -14582.404} C_VEL
LIN {X 0,Y 333.966,Z 264.382,A -85,B 0,C 180,E1 -14586.586,E2 -14586.586} C_VEL
LIN {X 0,Y 333.806,Z 264.404,A -85,B 0,C 180,E1 -14589.689,E2 -14589.689} C_VEL
LIN {X 0,Y 333.776,Z 264.41,A -85,B 0,C 180,E1 -14593.384,E2 -14593.384} C_VEL
LIN {X 0,Y 333.699,Z 264.42,A -85,B 0,C 180,E1 -14597.14,E2 -14597.14} C_VEL
LIN {X 0,Y 333.666,Z 264.419,A -85,B 0,C 180,E1 -14599.686,E2 -14599.686} C_VEL
LIN {X 0,Y 333.644,Z 264.422,A -85,B 0,C 180,E1 -14603.583,E2 -14603.583} C_VEL
LIN {X 0,Y 333.707,Z 264.414,A -85,B 0,C 180,E1 -14606.239,E2 -14606.239} C_VEL
LIN {X 0,Y 333.66,Z 264.424,A -85,B 0,C 180,E1 -14608.967,E2 -14608.967} C_VEL
LIN {X 0,Y 333.61,Z 264.431,A -85,B 0,C 180,E1 -14612.58,E2 -14612.58} C_VEL
LIN {X 0,Y 333.64,Z 264.424,A -85,B 0,C 180,E1 -14616.132,E2 -14616.132} C_VEL
LIN {X 0,Y 333.643,Z 264.423,A -85,B 0,C 180,E1 -14619.181,E2 -14619.181} C_VEL
LIN {X 0,Y 333.662,Z 264.425,A -85,B 0,C 180,E1 -14622.507,E2 -14622.507} C_VEL
LIN {X 0,Y 333.685,Z 264.419,A -85,B 0,C 180,E1 -14625.971,E2 -14625.971} C_VEL
LIN {X 0,Y 333.656,Z 264.42,A -85,B 0,C 180,E1 -14629.299,E2 -14629.299} C_VEL
LIN {X 0,Y 333.617,Z 264.425,A -85,B 0,C 180,E1 -14633.163,E2 -14633.163} C_VEL
LIN {X 0,Y 333.591,Z 264.429,A -85,B 0,C 180,E1 -14636.787,E2 -14636.787} C_VEL
LIN {X 0,Y 333.652,Z 264.425,A -85,B 0,C 180,E1 -14639.705,E2 -14639.705} C_VEL
LIN {X 0,Y 333.69,Z 264.418,A -85,B 0,C 180,E1 -14642.397,E2 -14642.397} C_VEL
LIN {X 0,Y 333.705,Z 264.416,A -85,B 0,C 180,E1 -14645.089,E2 -14645.089} C_VEL
LIN {X 0,Y 333.674,Z 264.433,A -85,B 0,C 180,E1 -14648.774,E2 -14648.774} C_VEL
LIN {X 0,Y 334.576,Z 267.103,A -85,B 0,C 180,E1 -14648.985,E2 -14648.985} C_VEL
LIN {X 0,Y 336.918,Z 269.959,A -85,B 0,C 180,E1 -14649.425,E2 -14649.425} C_VEL
LIN {X 0,Y 339.295,Z 273.381,A -85,B 0,C 180,E1 -14649.895,E2 -14649.895} C_VEL
LIN {X 0,Y 340.666,Z 274.987,A -85,B 0,C 180,E1 -14650.164,E2 -14650.164} C_VEL
LIN {X 0,Y 343.626,Z 278.698,A -85,B 0,C 180,E1 -14650.768,E2 -14650.768} C_VEL
LIN {X 0,Y 345.636,Z 281.158,A -85,B 0,C 180,E1 -14651.188,E2 -14651.188} C_VEL
LIN {X 0,Y 348.981,Z 284.821,A -85,B 0,C 180,E1 -14651.912,E2 -14651.912} C_VEL
LIN {X 0,Y 353.645,Z 290.015,A -85,B 0,C 180,E1 -14652.974,E2 -14652.974} C_VEL
LIN {X 0,Y 355.99,Z 292.311,A -85,B 0,C 180,E1 -14653.534,E2 -14653.534} C_VEL
LIN {X 0,Y 359.697,Z 296.219,A -85,B 0,C 180,E1 -14654.475,E2 -14654.475} C_VEL
LIN {X 0,Y 362.588,Z 298.707,A -85,B 0,C 180,E1 -14655.235,E2 -14655.235} C_VEL
LIN {X 0,Y 366.402,Z 302.663,A -85,B 0,C 180,E1 -14656.362,E2 -14656.362} C_VEL
LIN {X 0,Y 370.074,Z 305.646,A -85,B 0,C 180,E1 -14657.514,E2 -14657.514} C_VEL
LIN {X 0,Y 373.316,Z 309.04,A -85,B 0,C 180,E1 -14658.707,E2 -14658.707} C_VEL
LIN {X 0,Y 377.024,Z 311.666,A -85,B 0,C 180,E1 -14660.139,E2 -14660.139} C_VEL
LIN {X 0,Y 378.611,Z 312.684,A -85,B 0,C 180,E1 -14660.823,E2 -14660.823} C_VEL
LIN {X 0,Y 381.548,Z 316.027,A -85,B 0,C 180,E1 -14662.44,E2 -14662.44} C_VEL
LIN {X 0,Y 384.156,Z 318.092,A -85,B 0,C 180,E1 -14664.111,E2 -14664.111} C_VEL
LIN {X 0,Y 386.272,Z 319.183,A -85,B 0,C 180,E1 -14665.827,E2 -14665.827} C_VEL
LIN {X 0,Y 387.666,Z 319.541,A -85,B 0,C 180,E1 -14667.402,E2 -14667.402} C_VEL
LIN {X 0,Y 388.415,Z 319.649,A -85,B 0,C 180,E1 -14668.963,E2 -14668.963} C_VEL
LIN {X 0,Y 388.568,Z 319.676,A -85,B 0,C 180,E1 -14670,E2 -14670} C_VEL
LIN {X 0,Y 388.405,Z 319.646,A -85,B 0,C 180,E1 -14671.037,E2 -14671.037} C_VEL
LIN {X 0,Y 387.268,Z 319.401,A -85,B 0,C 180,E1 -14673.121,E2 -14673.121} C_VEL
LIN {X 0,Y 385.31,Z 318.794,A -85,B 0,C 180,E1 -14674.994,E2 -14674.994} C_VEL
LIN {X 0,Y 382.702,Z 317.099,A -85,B 0,C 180,E1 -14676.851,E2 -14676.851} C_VEL
